// TwinCAT 3 PLC project TcoCognexVision
// Title: TcoCognexVision
// Company: Vortex.Library
// ProjectVersion: 0.6.0.913
// ProgramVersion: 3.1.4023.0
// libraries:
//   Tc2_Standard, * (Beckhoff Automation GmbH)
//   Tc2_System, * (Beckhoff Automation GmbH)
//   Tc3_Module, * (Beckhoff Automation GmbH)
//   TcoAbstractions, 0.6.0.913 (Vortex.Library)
//   TcoCore, 0.6.0.913 (Vortex.Library)
//   TcoIo, 0.6.0.913 (Vortex.Library)
//   TcoUtilities, 0.6.0.913 (Vortex.Library)
// project tree:
//   / PlcTask.TcTTO
//   POUs/TcoDataman/v_5_x_x/IO/ TcoDatamanAcquisitionControl_v_5_x_x.TcDUT, TcoDatamanAcquisitionStatus_v_5_x_x.TcDUT, TcoDatamanIO_v_5_x_x.TcDUT, TcoDatamanResultData_v_5_x_x.TcDUT, TcoDatamanResultsControl_v_5_x_x.TcDUT, TcoDatamanResultsStatus_v_5_x_x.TcDUT, TcoDatamanSoftEventControl_v_5_x_x.TcDUT, TcoDatamanUserData_v_5_x_x.TcDUT
//   POUs/TcoDataman/v_5_x_x/Structs/ eDatamanResultDataSize_v_5_x_x.TcDUT, eDatamanUserDataSize_v_5_x_x.TcDUT, TcoDatamanConfig_v_5_x_x.TcDUT, TcoDatamanResults_v_5_x_x.TcDUT, TcoDatamanSignalStates_v_5_x_x.TcDUT, TcoDatamanStatus_v_5_x_x.TcDUT, TcoDatamanUser_v_5_x_x.TcDUT
//   POUs/TcoDataman/v_5_x_x/Tasks/ TcoDatamanClearResultData_v_5_x_x.TcPOU, TcoDatamanRead_v_5_x_x.TcPOU
//   POUs/TcoDataman/v_5_x_x/ TcoDataman_v_5_x_x.TcPOU
//   POUs/TcoDesigner/Structs/ eTcoDesignerTriggerType.TcDUT, TcoDesignerConfig_v_2_x_x.TcDUT, TcoDesignerData_2_x_x.TcDUT, TcoDesignerRootContainer.TcPOU, TcoDesignerStatus_v_2_x_x.TcDUT, TcoDesignerGenericResults_v_2_x_x.TcDUT, TcoDesignerPcToPlc_v_2_x_x.TcDUT, TcoDesignerPlcToPc_v_2_x_x.TcDUT
//   POUs/TcoDesigner/Tasks/ TcoDesignerTrigger_v_2_x_x.TcPOU, TcoDesignerClearInspectionResults_v_2_x_x.TcPOU
//   POUs/TcoDesigner/ TcoDesigner_v_2_x_x.TcPOU
//   POUs/TcoInsight/v_5_x_x/IO/ TcoInsightAcquisitionControl_v_5_x_x.TcDUT, TcoInsightAcquisitionStatus_v_5_x_x.TcDUT, TcoInsightIO_v_5_x_x.TcDUT, TcoInsightResultData_v_5_x_x.TcDUT, TcoInsightInspectionControl_v_5_x_x.TcDUT, TcoInsightInspectionStatus_v_5_x_x.TcDUT, TcoInsightSoftEventControl_v_5_x_x.TcDUT, TcoInsightCommandControl_v_5_x_x.TcDUT, TcoInsightUserData_v_5_x_x.TcDUT
//   POUs/TcoInsight/v_5_x_x/Structs/ eTcoInsightResultDataSize_v_5_x_x.TcDUT, eTcoInsightUserDataSize_v_5_x_x.TcDUT, TcoInsightConfig_v_5_x_x.TcDUT, TcoInsightResults_v_5_x_x.TcDUT, TcoInsightSignalStates_v_5_x_x.TcDUT, TcoInsightStatus_v_5_x_x.TcDUT, TcoInsightUser_v_5_x_x.TcDUT
//   POUs/TcoInsight/v_5_x_x/Tasks/ TcoInsightTrigger_v_5_x_x.TcPOU, TcoInsightChangeJobByName_v_5_x_x.TcPOU, TcoInsightChangeJobByNumber_v_5_x_x.TcPOU, TcoInsightClearInspectionResults_v_5_x_x.TcPOU, TcoInsightSoftEvent_v_5_x_x.TcPOU
//   POUs/TcoInsight/v_5_x_x/ TcoInsight_v_5_x_x.TcPOU
//   POUs/ TcoVisionParams.TcGVL
// real-time tasks:
//   TASK PlcTask: cycle T#10ms, priority 20, ADS port 350
//   TASK PNIO: cycle T#8ms, priority 21, ADS port 351
// I/O:
//   DEVICE Device 1 (Profinet Controller) (disabled), AmsNetId 172.20.10.104.2.1
//     dm260 [Cognex DataMan 260 ID Reader DMR-260#-#0]
//       modules: DAP_Module, Acquisition_Control, Acquisition_Status, Results_Control, Results_Status, Soft_Event_Control, User_Data_64_bytes, Result_Data_64_bytes
//     dm8700 [Cognex DataMan 8700 ID Reader CC-B DMR-87xx-xx]
//       modules: DAP_Module, Acquisition_Control, Acquisition_Status, Results_Control, Results_Status, Soft_Event_Control, User_Data_64_bytes, Result_Data_64_bytes
// variable links:
//   TcoCognexVision/TcoCognexVision Instance <-> Device 1 (Profinet Controller)/dm260
//     PlcTask Inputs/IO.dm260.AcquisitionStatus.Acquiring <-> API/Acquisition_Status/Acquisition_Status/Inputs/Acquisition_Status_Register/Acquiring
//     PlcTask Inputs/IO.dm260.AcquisitionStatus.MissedAcquisition <-> API/Acquisition_Status/Acquisition_Status/Inputs/Acquisition_Status_Register/Missed_Acquisition
//     PlcTask Inputs/IO.dm260.AcquisitionStatus.TriggerAcknowledge <-> API/Acquisition_Status/Acquisition_Status/Inputs/Acquisition_Status_Register/Trigger_Acknowledge
//     PlcTask Inputs/IO.dm260.AcquisitionStatus.TriggerID <-> API/Acquisition_Status/Acquisition_Status/Inputs/Trigger_ID
//     PlcTask Inputs/IO.dm260.AcquisitionStatus.TriggerReady <-> API/Acquisition_Status/Acquisition_Status/Inputs/Acquisition_Status_Register/Trigger_Ready
//     PlcTask Inputs/IO.dm260.PnIoBoxDiag <-> Inputs/PnIoBoxDiag
//     PlcTask Inputs/IO.dm260.PnIoBoxState <-> Inputs/PnIoBoxState
//     PlcTask Inputs/IO.dm260.ResultData.ResultCode <-> API/Result_Data_64_bytes/Result_Data_64_bytes/Inputs/Result_Code
//     PlcTask Inputs/IO.dm260.ResultData.ResultData <-> API/Result_Data_64_bytes/Result_Data_64_bytes/Inputs/Result_Data
//     PlcTask Inputs/IO.dm260.ResultData.ResultExtended <-> API/Result_Data_64_bytes/Result_Data_64_bytes/Inputs/Result_Extended
//     PlcTask Inputs/IO.dm260.ResultData.ResultID <-> API/Result_Data_64_bytes/Result_Data_64_bytes/Inputs/Result_ID
//     PlcTask Inputs/IO.dm260.ResultData.ResultLength <-> API/Result_Data_64_bytes/Result_Data_64_bytes/Inputs/Result_Length
//     PlcTask Inputs/IO.dm260.ResultsStatus.DecodeComplete <-> API/Results_Status/Results_Status/Inputs/Results_Status_Register/Decode_Complete
//     PlcTask Inputs/IO.dm260.ResultsStatus.Decoding <-> API/Results_Status/Results_Status/Inputs/Results_Status_Register/Decoding
//     PlcTask Inputs/IO.dm260.ResultsStatus.ErrorDetected <-> API/Results_Status/Results_Status/Inputs/Results_Status_Register/Set_when_reader_fault_occurs
//     PlcTask Inputs/IO.dm260.ResultsStatus.ResultsAvailable <-> API/Results_Status/Results_Status/Inputs/Results_Status_Register/Results_Available
//     PlcTask Inputs/IO.dm260.ResultsStatus.ResultsBufferOverrun <-> API/Results_Status/Results_Status/Inputs/Results_Status_Register/Results_Buffer_Overrun
//     PlcTask Inputs/IO.dm260.SoftEventControl.ExecuteDMCCAcknowledge <-> API/Soft_Event_Control/Soft_Event_Control/Inputs/Soft_Event_Acknowledge_Register/Execute_DMCC_Acknowledge
//     PlcTask Inputs/IO.dm260.SoftEventControl.SetMatchStringAcknowledge <-> API/Soft_Event_Control/Soft_Event_Control/Inputs/Soft_Event_Acknowledge_Register/Set_Match_String_Acknowledge
//     PlcTask Inputs/IO.dm260.SoftEventControl.TrainBrightnessAcknowledge <-> API/Soft_Event_Control/Soft_Event_Control/Inputs/Soft_Event_Acknowledge_Register/Train_Brightness_Acknowledge
//     PlcTask Inputs/IO.dm260.SoftEventControl.TrainCodeAcknowledge <-> API/Soft_Event_Control/Soft_Event_Control/Inputs/Soft_Event_Acknowledge_Register/Train_Code_Acknowledge
//     PlcTask Inputs/IO.dm260.SoftEventControl.TrainFocusAcknowledge <-> API/Soft_Event_Control/Soft_Event_Control/Inputs/Soft_Event_Acknowledge_Register/Train_Focus_Acknowledge
//     PlcTask Inputs/IO.dm260.SoftEventControl.TrainMatchStringAcknowledge <-> API/Soft_Event_Control/Soft_Event_Control/Inputs/Soft_Event_Acknowledge_Register/Train_Match_String_Acknowledge
//     PlcTask Inputs/IO.dm260.SoftEventControl.UntrainAcknowledge <-> API/Soft_Event_Control/Soft_Event_Control/Inputs/Soft_Event_Acknowledge_Register/Untrain_Acknowledge
//     PlcTask Outputs/IO.dm260.AcquisitionControl.Trigger <-> API/Acquisition_Control/Acquisition_Control/Outputs/Acquisition_Control_Register/Trigger
//     PlcTask Outputs/IO.dm260.AcquisitionControl.TriggerEnable <-> API/Acquisition_Control/Acquisition_Control/Outputs/Acquisition_Control_Register/Trigger_Enable
//     PlcTask Outputs/IO.dm260.PnIoBoxCtrl <-> Outputs/PnIoBoxCtrl
//     PlcTask Outputs/IO.dm260.ResultsControl.EnableResultBuffering <-> API/Results_Control/Results_Control/Outputs/Results_Control_Register/Enable_Result_Buffering
//     PlcTask Outputs/IO.dm260.ResultsControl.ResultsAcknowledge <-> API/Results_Control/Results_Control/Outputs/Results_Control_Register/Results_Acknowledge
//     PlcTask Outputs/IO.dm260.SoftEventControl.ExecuteDMCC <-> API/Soft_Event_Control/Soft_Event_Control/Outputs/Soft_Event_Control_Register/Execute_DMCC
//     PlcTask Outputs/IO.dm260.SoftEventControl.SetMatchString <-> API/Soft_Event_Control/Soft_Event_Control/Outputs/Soft_Event_Control_Register/Set_Match_String
//     PlcTask Outputs/IO.dm260.SoftEventControl.TrainBrightness <-> API/Soft_Event_Control/Soft_Event_Control/Outputs/Soft_Event_Control_Register/Train_Brightness
//     PlcTask Outputs/IO.dm260.SoftEventControl.TrainCode <-> API/Soft_Event_Control/Soft_Event_Control/Outputs/Soft_Event_Control_Register/Train_Code
//     PlcTask Outputs/IO.dm260.SoftEventControl.TrainFocus <-> API/Soft_Event_Control/Soft_Event_Control/Outputs/Soft_Event_Control_Register/Train_Focus
//     PlcTask Outputs/IO.dm260.SoftEventControl.TrainMatchString <-> API/Soft_Event_Control/Soft_Event_Control/Outputs/Soft_Event_Control_Register/Train_Match_String
//     PlcTask Outputs/IO.dm260.SoftEventControl.Untrain <-> API/Soft_Event_Control/Soft_Event_Control/Outputs/Soft_Event_Control_Register/Untrain
//     PlcTask Outputs/IO.dm260.UserData.UserData <-> API/User_Data_64_bytes/User_Data_64_bytes/Outputs/User_Data
//     PlcTask Outputs/IO.dm260.UserData.UserDataLength <-> API/User_Data_64_bytes/User_Data_64_bytes/Outputs/User_Data_Length
//     PlcTask Outputs/IO.dm260.UserData.UserDataOption <-> API/User_Data_64_bytes/User_Data_64_bytes/Outputs/User_Data_Option
//   TcoCognexVision/TcoCognexVision Instance <-> Device 1 (Profinet Controller)/dm8700
//     PlcTask Inputs/IO.dm8700.AcquisitionStatus.Acquiring <-> API/Acquisition_Status/Acquisition_Status/Inputs/Acquisition_Status_Register/Acquiring
//     PlcTask Inputs/IO.dm8700.AcquisitionStatus.MissedAcquisition <-> API/Acquisition_Status/Acquisition_Status/Inputs/Acquisition_Status_Register/Missed_Acquisition
//     PlcTask Inputs/IO.dm8700.AcquisitionStatus.TriggerAcknowledge <-> API/Acquisition_Status/Acquisition_Status/Inputs/Acquisition_Status_Register/Trigger_Acknowledge
//     PlcTask Inputs/IO.dm8700.AcquisitionStatus.TriggerID <-> API/Acquisition_Status/Acquisition_Status/Inputs/Trigger_ID
//     PlcTask Inputs/IO.dm8700.AcquisitionStatus.TriggerReady <-> API/Acquisition_Status/Acquisition_Status/Inputs/Acquisition_Status_Register/Trigger_Ready
//     PlcTask Inputs/IO.dm8700.PnIoBoxDiag <-> Inputs/PnIoBoxDiag
//     PlcTask Inputs/IO.dm8700.PnIoBoxState <-> Inputs/PnIoBoxState
//     PlcTask Inputs/IO.dm8700.ResultData.ResultCode <-> API/Result_Data_64_bytes/Result_Data_64_bytes/Inputs/Result_Code
//     PlcTask Inputs/IO.dm8700.ResultData.ResultData <-> API/Result_Data_64_bytes/Result_Data_64_bytes/Inputs/Result_Data
//     PlcTask Inputs/IO.dm8700.ResultData.ResultExtended <-> API/Result_Data_64_bytes/Result_Data_64_bytes/Inputs/Result_Extended
//     PlcTask Inputs/IO.dm8700.ResultData.ResultID <-> API/Result_Data_64_bytes/Result_Data_64_bytes/Inputs/Result_ID
//     PlcTask Inputs/IO.dm8700.ResultData.ResultLength <-> API/Result_Data_64_bytes/Result_Data_64_bytes/Inputs/Result_Length
//     PlcTask Inputs/IO.dm8700.ResultsStatus.DecodeComplete <-> API/Results_Status/Results_Status/Inputs/Results_Status_Register/Decode_Complete
//     PlcTask Inputs/IO.dm8700.ResultsStatus.Decoding <-> API/Results_Status/Results_Status/Inputs/Results_Status_Register/Decoding
//     PlcTask Inputs/IO.dm8700.ResultsStatus.ErrorDetected <-> API/Results_Status/Results_Status/Inputs/Results_Status_Register/Set_when_reader_fault_occurs
//     PlcTask Inputs/IO.dm8700.ResultsStatus.ResultsAvailable <-> API/Results_Status/Results_Status/Inputs/Results_Status_Register/Results_Available
//     PlcTask Inputs/IO.dm8700.ResultsStatus.ResultsBufferOverrun <-> API/Results_Status/Results_Status/Inputs/Results_Status_Register/Results_Buffer_Overrun
//     PlcTask Inputs/IO.dm8700.SoftEventControl.ExecuteDMCCAcknowledge <-> API/Soft_Event_Control/Soft_Event_Control/Inputs/Soft_Event_Acknowledge_Register/Execute_DMCC_Acknowledge
//     PlcTask Inputs/IO.dm8700.SoftEventControl.SetMatchStringAcknowledge <-> API/Soft_Event_Control/Soft_Event_Control/Inputs/Soft_Event_Acknowledge_Register/Set_Match_String_Acknowledge
//     PlcTask Inputs/IO.dm8700.SoftEventControl.TrainBrightnessAcknowledge <-> API/Soft_Event_Control/Soft_Event_Control/Inputs/Soft_Event_Acknowledge_Register/Train_Brightness_Acknowledge
//     PlcTask Inputs/IO.dm8700.SoftEventControl.TrainCodeAcknowledge <-> API/Soft_Event_Control/Soft_Event_Control/Inputs/Soft_Event_Acknowledge_Register/Train_Code_Acknowledge
//     PlcTask Inputs/IO.dm8700.SoftEventControl.TrainFocusAcknowledge <-> API/Soft_Event_Control/Soft_Event_Control/Inputs/Soft_Event_Acknowledge_Register/Train_Focus_Acknowledge
//     PlcTask Inputs/IO.dm8700.SoftEventControl.TrainMatchStringAcknowledge <-> API/Soft_Event_Control/Soft_Event_Control/Inputs/Soft_Event_Acknowledge_Register/Train_Match_String_Acknowledge
//     PlcTask Inputs/IO.dm8700.SoftEventControl.UntrainAcknowledge <-> API/Soft_Event_Control/Soft_Event_Control/Inputs/Soft_Event_Acknowledge_Register/Untrain_Acknowledge
//     PlcTask Outputs/IO.dm8700.AcquisitionControl.Trigger <-> API/Acquisition_Control/Acquisition_Control/Outputs/Acquisition_Control_Register/Trigger
//     PlcTask Outputs/IO.dm8700.AcquisitionControl.TriggerEnable <-> API/Acquisition_Control/Acquisition_Control/Outputs/Acquisition_Control_Register/Trigger_Enable
//     PlcTask Outputs/IO.dm8700.PnIoBoxCtrl <-> Outputs/PnIoBoxCtrl
//     PlcTask Outputs/IO.dm8700.ResultsControl.EnableResultBuffering <-> API/Results_Control/Results_Control/Outputs/Results_Control_Register/Enable_Result_Buffering
//     PlcTask Outputs/IO.dm8700.ResultsControl.ResultsAcknowledge <-> API/Results_Control/Results_Control/Outputs/Results_Control_Register/Results_Acknowledge
//     PlcTask Outputs/IO.dm8700.SoftEventControl.ExecuteDMCC <-> API/Soft_Event_Control/Soft_Event_Control/Outputs/Soft_Event_Control_Register/Execute_DMCC
//     PlcTask Outputs/IO.dm8700.SoftEventControl.SetMatchString <-> API/Soft_Event_Control/Soft_Event_Control/Outputs/Soft_Event_Control_Register/Set_Match_String
//     PlcTask Outputs/IO.dm8700.SoftEventControl.TrainBrightness <-> API/Soft_Event_Control/Soft_Event_Control/Outputs/Soft_Event_Control_Register/Train_Brightness
//     PlcTask Outputs/IO.dm8700.SoftEventControl.TrainCode <-> API/Soft_Event_Control/Soft_Event_Control/Outputs/Soft_Event_Control_Register/Train_Code
//     PlcTask Outputs/IO.dm8700.SoftEventControl.TrainFocus <-> API/Soft_Event_Control/Soft_Event_Control/Outputs/Soft_Event_Control_Register/Train_Focus
//     PlcTask Outputs/IO.dm8700.SoftEventControl.TrainMatchString <-> API/Soft_Event_Control/Soft_Event_Control/Outputs/Soft_Event_Control_Register/Train_Match_String
//     PlcTask Outputs/IO.dm8700.SoftEventControl.Untrain <-> API/Soft_Event_Control/Soft_Event_Control/Outputs/Soft_Event_Control_Register/Untrain
//     PlcTask Outputs/IO.dm8700.UserData.UserData <-> API/User_Data_64_bytes/User_Data_64_bytes/Outputs/User_Data
//     PlcTask Outputs/IO.dm8700.UserData.UserDataLength <-> API/User_Data_64_bytes/User_Data_64_bytes/Outputs/User_Data_Length
//     PlcTask Outputs/IO.dm8700.UserData.UserDataOption <-> API/User_Data_64_bytes/User_Data_64_bytes/Outputs/User_Data_Option

CONFIGURATION TcoCognexVision
    RESOURCE PLC ON TwinCAT3
        TASK PlcTask(INTERVAL := T#10ms, PRIORITY := 20);
        PROGRAM MAIN WITH PlcTask : MAIN;
    END_RESOURCE
END_CONFIGURATION

// ---- POUs/TcoDataman/v_5_x_x/IO/TcoDatamanAcquisitionControl_v_5_x_x.TcDUT
TYPE TcoDatamanAcquisitionControl_v_5_x_x :
STRUCT
    TriggerEnable AT %Q* : BOOL;
    Trigger AT %Q* : BOOL;
END_STRUCT
END_TYPE

// ---- POUs/TcoDataman/v_5_x_x/IO/TcoDatamanAcquisitionStatus_v_5_x_x.TcDUT
TYPE TcoDatamanAcquisitionStatus_v_5_x_x :
STRUCT
    TriggerReady AT %I* : BOOL;
    TriggerAcknowledge AT %I* : BOOL;
    Acquiring AT %I* : BOOL;
    MissedAcquisition AT %I* : BOOL;
    TriggerID AT %I* : UINT;
END_STRUCT
END_TYPE

// ---- POUs/TcoDataman/v_5_x_x/IO/TcoDatamanIO_v_5_x_x.TcDUT
TYPE TcoDatamanIO_v_5_x_x :
STRUCT
    PnIoBoxState AT %I* : UINT;
    PnIoBoxDiag AT %I* : UINT;
    PnIoBoxCtrl AT %Q* : UINT;
    AcquisitionControl : TcoDatamanAcquisitionControl_v_5_x_x;
    AcquisitionStatus : TcoDatamanAcquisitionStatus_v_5_x_x;
    ResultsControl : TcoDatamanResultsControl_v_5_x_x;
    ResultsStatus : TcoDatamanResultsStatus_v_5_x_x;
    SoftEventControl : TcoDatamanSoftEventControl_v_5_x_x;
    UserData : TcoDatamanUserData_v_5_x_x;
    ResultData : TcoDatamanResultData_v_5_x_x;
END_STRUCT
END_TYPE

// ---- POUs/TcoDataman/v_5_x_x/IO/TcoDatamanResultData_v_5_x_x.TcDUT
TYPE TcoDatamanResultData_v_5_x_x :
STRUCT
    ResultID AT %I* : UINT;
    ResultCode AT %I* : UINT;
    ResultExtended AT %I* : UINT;
    ResultLength AT %I* : UINT;
    ResultData AT %I* : ARRAY[0..245] OF BYTE;
END_STRUCT
END_TYPE

// ---- POUs/TcoDataman/v_5_x_x/IO/TcoDatamanResultsControl_v_5_x_x.TcDUT
TYPE TcoDatamanResultsControl_v_5_x_x :
STRUCT
    EnableResultBuffering AT %Q* : BOOL;
    ResultsAcknowledge AT %Q* : BOOL;
END_STRUCT
END_TYPE

// ---- POUs/TcoDataman/v_5_x_x/IO/TcoDatamanResultsStatus_v_5_x_x.TcDUT
TYPE TcoDatamanResultsStatus_v_5_x_x :
STRUCT
    Decoding AT %I* : BOOL;
    DecodeComplete AT %I* : BOOL;
    ResultsBufferOverrun AT %I* : BOOL;
    ResultsAvailable AT %I* : BOOL;
    ErrorDetected AT %I* : BOOL;
END_STRUCT
END_TYPE

// ---- POUs/TcoDataman/v_5_x_x/IO/TcoDatamanSoftEventControl_v_5_x_x.TcDUT
TYPE TcoDatamanSoftEventControl_v_5_x_x :
STRUCT
    TrainCodeAcknowledge AT %I* : BOOL;
    TrainMatchStringAcknowledge AT %I* : BOOL;
    TrainFocusAcknowledge AT %I* : BOOL;
    TrainBrightnessAcknowledge AT %I* : BOOL;
    UntrainAcknowledge AT %I* : BOOL;
    Reserved05 AT %I* : BOOL;
    ExecuteDMCCAcknowledge AT %I* : BOOL;
    SetMatchStringAcknowledge AT %I* : BOOL;
    TrainCode AT %Q* : BOOL;
    TrainMatchString AT %Q* : BOOL;
    TrainFocus AT %Q* : BOOL;
    TrainBrightness AT %Q* : BOOL;
    Untrain AT %Q* : BOOL;
    Reserved15 AT %Q* : BOOL;
    ExecuteDMCC AT %Q* : BOOL;
    SetMatchString AT %Q* : BOOL;
END_STRUCT
END_TYPE

// ---- POUs/TcoDataman/v_5_x_x/IO/TcoDatamanUserData_v_5_x_x.TcDUT
TYPE TcoDatamanUserData_v_5_x_x :
STRUCT
    UserDataOption AT %Q* : UINT;
    UserDataLength AT %Q* : UINT;
    UserData AT %Q* : ARRAY[0..249] OF BYTE;
END_STRUCT
END_TYPE

// ---- POUs/TcoDataman/v_5_x_x/Structs/eDatamanResultDataSize_v_5_x_x.TcDUT
{attribute 'qualified_only'}
{attribute 'strict'}
TYPE eDatamanResultDataSize_v_5_x_x :
(
    RESULT_DATA_16B := 16,
    RESULT_DATA_32B := 32,
    RESULT_DATA_64B := 64,
    RESULT_DATA_128B := 128,
    RESULT_DATA_246B := 246
);
END_TYPE

// ---- POUs/TcoDataman/v_5_x_x/Structs/eDatamanUserDataSize_v_5_x_x.TcDUT
{attribute 'qualified_only'}
{attribute 'strict'}
TYPE eDatamanUserDataSize_v_5_x_x :
(
    USER_DATA_16B := 16,
    USER_DATA_32B := 32,
    USER_DATA_64B := 64,
    USER_DATA_128B := 128,
    USER_DATA_250B := 250
);
END_TYPE

// ---- POUs/TcoDataman/v_5_x_x/Structs/TcoDatamanConfig_v_5_x_x.TcDUT
TYPE TcoDatamanConfig_v_5_x_x :
STRUCT
    ResultDataSize : eDatamanResultDataSize_v_5_x_x := eDatamanResultDataSize_v_5_x_x.RESULT_DATA_64B;
    UserDataSize : eDatamanUserDataSize_v_5_x_x := eDatamanUserDataSize_v_5_x_x.USER_DATA_64B;
    DataFormat : eTcoDataFormat := TcoUtilities.eTcoDataFormat.BigEndian;
    ContinuousReading : BOOL := FALSE;
    UpdateStatesPermanently : BOOL := FALSE;
    InfoTime : TIME := T#2S;
    ErrorTime : TIME := T#5S;
    ShowUserData : BOOL := FALSE;
    ShowResultsData : BOOL := FALSE;
END_STRUCT
END_TYPE

// ---- POUs/TcoDataman/v_5_x_x/Structs/TcoDatamanResults_v_5_x_x.TcDUT
TYPE TcoDatamanResults_v_5_x_x :
STRUCT
    Id : UINT;
    Code : UINT;
    Extended : UINT;
    Length : UINT;
    Data : ARRAY[0..TcoVisionParams.MAX_BYTE_ARRAY] OF BYTE;
END_STRUCT
END_TYPE

// ---- POUs/TcoDataman/v_5_x_x/Structs/TcoDatamanSignalStates_v_5_x_x.TcDUT
{attribute addProperty Name "Signal states"}
{attribute wpf [Container(Layout.Stack)]}
TYPE TcoDatamanSignalStates_v_5_x_x :
STRUCT
    {attribute wpf [Container(Layout.Stack,"Acquisition control")]}
    {attribute wpf [Group(Layout.GroupBox)]}
    {attribute addProperty Name "<#Trigger enable#>"}
    TriggerEnable : BOOL;
    {attribute addProperty Name "<#Trigger#>"}
    Trigger : BOOL;
    {attribute wpf [Container(Layout.Stack,"Result control")]}
    {attribute wpf [Group(Layout.GroupBox)]}
    {attribute addProperty Name "<#Enable result buffering#>"}
    EnableResultBuffering : BOOL;
    {attribute addProperty Name "<#Result acknowledge#>"}
    ResultsAcknowledge : BOOL;
    {attribute wpf [Container(Layout.Stack,"Acquisition status")]}
    {attribute wpf [Group(Layout.GroupBox)]}
    {attribute addProperty Name "<#Trigger ready#>"}
    TriggerReady : BOOL;
    {attribute addProperty Name "<#Trigger acknowledge#>"}
    TriggerAcknowledge : BOOL;
    {attribute addProperty Name "<#Acquiring#>"}
    Acquiring : BOOL;
    {attribute addProperty Name "<#Missed acquisition#>"}
    MissedAcquisition : BOOL;
    {attribute addProperty Name "<#Trigger ID#>"}
    TriggerID : UINT;
    {attribute wpf [Container(Layout.Stack,"Result status")]}
    {attribute wpf [Group(Layout.GroupBox)]}
    {attribute addProperty Name "<#Decoding#>"}
    Decoding : BOOL;
    {attribute addProperty Name "<#Decode complete#>"}
    DecodeComplete : BOOL;
    {attribute addProperty Name "<#Result buffer overrun#>"}
    ResultsBufferOverrun : BOOL;
    {attribute addProperty Name "<#Results available#>"}
    ResultsAvailable : BOOL;
    {attribute addProperty Name "<#Error detected#>"}
    ErrorDetected : BOOL;
    {attribute wpf [Container(Layout.Stack,"Result data")]}
    {attribute wpf [Group(Layout.GroupBox)]}
    {attribute addProperty Name "<#Result ID#>"}
    ResultID : UINT;
    {attribute addProperty Name "<#Result code#>"}
    ResultCode : UINT;
    {attribute addProperty Name "<#Result extended#>"}
    ResultExtended : UINT;
    {attribute addProperty Name "<#Result length#>"}
    ResultLength : UINT;
END_STRUCT
END_TYPE

// ---- POUs/TcoDataman/v_5_x_x/Structs/TcoDatamanStatus_v_5_x_x.TcDUT
TYPE TcoDatamanStatus_v_5_x_x :
STRUCT
    ActionDescription : STRING(100);
    ResultString : STRING;
    SignalStatus : TcoDatamanSignalStates_v_5_x_x;
END_STRUCT
END_TYPE

// ---- POUs/TcoDataman/v_5_x_x/Structs/TcoDatamanUser_v_5_x_x.TcDUT
TYPE TcoDatamanUser_v_5_x_x :
STRUCT
    Option : UINT;
    Length : UINT;
    Data : ARRAY[0..TcoVisionParams.MAX_BYTE_ARRAY] OF BYTE;
END_STRUCT
END_TYPE

// ---- POUs/TcoDesigner/Structs/eTcoDesignerTriggerType.TcDUT
{attribute 'qualified_only'}
{attribute 'strict'}
TYPE eTcoDesignerTriggerType :
(
    Trigger := 0,
    TriggerFast := 1,
    TriggerWithTimeout := 2
);
END_TYPE

// ---- POUs/TcoDesigner/Structs/TcoDesignerConfig_v_2_x_x.TcDUT
TYPE TcoDesignerConfig_v_2_x_x :
STRUCT
    TriggerTimemout : TIME := T#15S;
    ConnectionTimemout : TIME := T#10S;
    InfoTime : TIME := T#2S;
    ErrorTime : TIME := T#5S;
END_STRUCT
END_TYPE

// ---- POUs/TcoDesigner/Structs/TcoDesignerData_2_x_x.TcDUT
{attribute wpf [Container(Layout.Stack)]}
TYPE TcoDesignerData_2_x_x :
STRUCT
    {attribute wpf [Container(Layout.Stack,"PcToPlc")]}
    {attribute addProperty Name "<#PCtoPLC#>"}
    PcToPlc : TcoDesignerPcToPlc_v_2_x_x;
    {attribute wpf [Container(Layout.Stack,"PlcToPc")]}
    {attribute addProperty Name "<#PLCtoPC#>"}
    PlcToPc : TcoDesignerPlcToPc_v_2_x_x;
END_STRUCT
END_TYPE

// ---- POUs/TcoDesigner/Structs/TcoDesignerStatus_v_2_x_x.TcDUT
TYPE TcoDesignerStatus_v_2_x_x :
STRUCT
    ActionDescription : STRING(100);
    ClientConnected : BOOL;
    {attribute wpf [Container(Layout.Stack,"PcToPlc")]}
    {attribute wpf [Group(Layout.GroupBox)]}
    SignalStatus : TcoDesignerPcToPlc_v_2_x_x;
END_STRUCT
END_TYPE

// ---- POUs/TcoDesigner/Structs/TcoDesignerGenericResults_v_2_x_x.TcDUT
TYPE TcoDesignerGenericResults_v_2_x_x :
STRUCT
    {attribute addProperty Name "<#GeneralResult Pass#>"}
    ResultPass : BOOL;
    {attribute addProperty Name "<#GeneralResult FAIL#>"}
    ResultFail : BOOL;
END_STRUCT
END_TYPE

// ---- POUs/TcoDesigner/Structs/TcoDesignerPcToPlc_v_2_x_x.TcDUT
{attribute wpf [Container(Layout.Stack)]}
TYPE TcoDesignerPcToPlc_v_2_x_x :
STRUCT
    {attribute wpf [Container(Layout.Stack,"State")]}
    {attribute addProperty Name "<#SystemOnline#>"}
    SystemOnline : BOOL; //indication that designer PC app and inspection are running
    {attribute addProperty Name "<#InspectionReady#>"}
    InspectionReady : BOOL; // inspection is ready
    {attribute addProperty Name "<#ResultsAvailable#>"}
    ResultsAvailable : BOOL; //results are available and valid
    {attribute addProperty Name "<#JobId#>"}
    JobId : UINT; // actual job id
    {attribute addProperty Name "<#JobName#>"}
    JobName : STRING; //aktual job name
    {attribute addProperty Name "<#JobLoadDone#>"}
    JobLoadDone : BOOL;
    {attribute addProperty Name "<#ClearResultsAck#>"}
    ClearResultsAck : BOOL;
    {attribute addProperty Name "<#Trigger Counter#>"}
    TriggerCounter : UDINT;
    {attribute addProperty Name "<#Error#>"}
    Error : BOOL;
    {attribute addProperty Name "<#LiveBit#>"}
    LiveBit : BOOL;
    {attribute addProperty Name "<#ErrorMsg#>"}
    ErrorMsg : STRING;
    {attribute addProperty Name "<#TriggerTimeout#>"}
    TriggerTimeout : BOOL;
    {attribute wpf [Container(Layout.Stack,"Results")]}
    {attribute addProperty Name "<#Results#>"}
    InspectionResults : TcoDesignerGenericResults_v_2_x_x;
END_STRUCT
END_TYPE

// ---- POUs/TcoDesigner/Structs/TcoDesignerPlcToPc_v_2_x_x.TcDUT
{attribute wpf [Container(Layout.Stack)]}
TYPE TcoDesignerPlcToPc_v_2_x_x :
STRUCT
    {attribute wpf [Container(Layout.Stack,"Control")]}
    {attribute addProperty Name "<#Trigger#>"}
    Trigger : BOOL;
    {attribute addProperty Name "<#ResultsAck#>"}
    ResultsAck : BOOL;
    {attribute addProperty Name "<#Reset#>"}
    Reset : BOOL;
    {attribute addProperty Name "<#JobLoadId#>"}
    JobLoadId : UINT;
    {attribute addProperty Name "<#LoadJob#>"}
    LoadJob : BOOL;
    {attribute addProperty Name "<#ClearResults#>"}
    ClearResults : BOOL;
    {attribute addProperty Name "<#Timeout[ms]#>"}
    Timeout : UINT;
    {attribute addProperty Name "<# PartId #>"}
    PartId : STRING; //napr. DMC Code
END_STRUCT
END_TYPE

// ---- POUs/TcoInsight/v_5_x_x/IO/TcoInsightAcquisitionControl_v_5_x_x.TcDUT
TYPE TcoInsightAcquisitionControl_v_5_x_x :
STRUCT
    AcquisitionTriggerEnable AT %Q* : BOOL;
    AcquisitionTrigger AT %Q* : BOOL;
    ClearExposureComplete AT %Q* : BOOL;
    SetOffline AT %Q* : BOOL;
END_STRUCT
END_TYPE

// ---- POUs/TcoInsight/v_5_x_x/IO/TcoInsightAcquisitionStatus_v_5_x_x.TcDUT
TYPE TcoInsightAcquisitionStatus_v_5_x_x :
STRUCT
    AcquisitionTriggerReady AT %I* : BOOL;
    AcquisitionTriggerAcknowledge AT %I* : BOOL;
    ExposureComplete AT %I* : BOOL;
    MissedAcquisition AT %I* : BOOL;
    OfflineReason0 AT %I* : BOOL;
    OfflineReason1 AT %I* : BOOL;
    OfflineReason2 AT %I* : BOOL;
    Online AT %I* : BOOL;
    AcquisitionID AT %I* : UINT;
END_STRUCT
END_TYPE

// ---- POUs/TcoInsight/v_5_x_x/IO/TcoInsightIO_v_5_x_x.TcDUT
TYPE TcoInsightIO_v_5_x_x :
STRUCT
    PnIoBoxState AT %I* : UINT;
    PnIoBoxDiag AT %I* : UINT;
    PnIoBoxCtrl AT %Q* : UINT;
    AcquisitionControl : TcoInsightAcquisitionControl_v_5_x_x;
    AcquisitionStatus : TcoInsightAcquisitionStatus_v_5_x_x;
    InspectionControl : TcoInsightInspectionControl_v_5_x_x;
    InspectionStatus : TcoInsightInspectionStatus_v_5_x_x;
    CommandControl : TcoInsightCommandControl_v_5_x_x;
    SoftEventControl : TcoInsightSoftEventControl_v_5_x_x;
    UserData : TcoInsightUserData_v_5_x_x;
    ResultsData : TcoInsightResultData_v_5_x_x;
END_STRUCT
END_TYPE

// ---- POUs/TcoInsight/v_5_x_x/IO/TcoInsightResultData_v_5_x_x.TcDUT
TYPE TcoInsightResultData_v_5_x_x :
STRUCT
    InspectionID AT %I* : UINT;
    ResultCode AT %I* : UINT;
    InspectionResults AT %I* : ARRAY[0..245] OF BYTE;
END_STRUCT
END_TYPE

// ---- POUs/TcoInsight/v_5_x_x/IO/TcoInsightInspectionControl_v_5_x_x.TcDUT
TYPE TcoInsightInspectionControl_v_5_x_x :
STRUCT
    EnableResultsBuffering AT %Q* : BOOL;
    AcknowledgeInspectionResults AT %Q* : BOOL;
    ExtendedUserDataSet AT %Q* : BOOL;
    ExecuteCommand AT %Q* : BOOL;
    ClearError AT %Q* : BOOL;
END_STRUCT
END_TYPE

// ---- POUs/TcoInsight/v_5_x_x/IO/TcoInsightInspectionStatus_v_5_x_x.TcDUT
TYPE TcoInsightInspectionStatus_v_5_x_x :
STRUCT
    SystemBusy AT %I* : BOOL;
    InspectionCompleted AT %I* : BOOL;
    ResultsBufferOverrun AT %I* : BOOL;
    ResultsValid AT %I* : BOOL;
    CommandExecuting AT %I* : BOOL;
    CommandComplete AT %I* : BOOL;
    CommandFailed AT %I* : BOOL;
    ExtendedUserDataSetAcknowledge AT %I* : BOOL;
    OverallJobPassFail AT %I* : BOOL;
    TestRunReady AT %I* : BOOL;
    Error AT %I* : BOOL;
    ErrorCode AT %I* : UINT;
END_STRUCT
END_TYPE

// ---- POUs/TcoInsight/v_5_x_x/IO/TcoInsightSoftEventControl_v_5_x_x.TcDUT
TYPE TcoInsightSoftEventControl_v_5_x_x :
STRUCT
    TriggerSoftEventAcknowledge AT %I* : ARRAY[0..7] OF BOOL;
    TriggerSoftEvent AT %Q* : ARRAY[0..7] OF BOOL;
END_STRUCT
END_TYPE

// ---- POUs/TcoInsight/v_5_x_x/IO/TcoInsightCommandControl_v_5_x_x.TcDUT
TYPE TcoInsightCommandControl_v_5_x_x :
STRUCT
    CurrentJobID AT %I* : UINT;
    Command AT %Q* : UINT;
END_STRUCT
END_TYPE

// ---- POUs/TcoInsight/v_5_x_x/IO/TcoInsightUserData_v_5_x_x.TcDUT
TYPE TcoInsightUserData_v_5_x_x :
STRUCT
    UserData AT %Q* : ARRAY[0..253] OF BYTE;
END_STRUCT
END_TYPE

// ---- POUs/TcoInsight/v_5_x_x/Structs/eTcoInsightResultDataSize_v_5_x_x.TcDUT
{attribute 'qualified_only'}
{attribute 'strict'}
TYPE eTcoInsightResultDataSize_v_5_x_x :
(
    RESULT_DATA_16B := 16,
    RESULT_DATA_32B := 32,
    RESULT_DATA_64B := 64,
    RESULT_DATA_128B := 128,
    RESULT_DATA_246B := 250
);
END_TYPE

// ---- POUs/TcoInsight/v_5_x_x/Structs/eTcoInsightUserDataSize_v_5_x_x.TcDUT
{attribute 'qualified_only'}
{attribute 'strict'}
TYPE eTcoInsightUserDataSize_v_5_x_x :
(
    USER_DATA_16B := 16,
    USER_DATA_32B := 32,
    USER_DATA_64B := 64,
    USER_DATA_128B := 128,
    USER_DATA_250B := 254
);
END_TYPE

// ---- POUs/TcoInsight/v_5_x_x/Structs/TcoInsightConfig_v_5_x_x.TcDUT
TYPE TcoInsightConfig_v_5_x_x :
STRUCT
    ResultDataSize : eTcoInsightResultDataSize_v_5_x_x := eTcoInsightResultDataSize_v_5_x_x.RESULT_DATA_64B;
    UserDataSize : eTcoInsightUserDataSize_v_5_x_x := eTcoInsightUserDataSize_v_5_x_x.USER_DATA_64B;
    DataFormat : eTcoDataFormat := TcoUtilities.eTcoDataFormat.BigEndian;
    UpdateStatesPermanently : BOOL := FALSE;
    MaxJobNumber : UINT := 999;
    InfoTime : TIME := T#2S;
    ErrorTime : TIME := T#5S;
    ShowUserData : BOOL := FALSE;
    ShowResultsData : BOOL := FALSE;
//	ServiceJobNumber		:	UINT;
//	ServiceJobName			:	STRING;
//	ServiceSoftEventNumber	:	UINT;
END_STRUCT
END_TYPE

// ---- POUs/TcoInsight/v_5_x_x/Structs/TcoInsightResults_v_5_x_x.TcDUT
TYPE TcoInsightResults_v_5_x_x :
STRUCT
    InspectionId : UINT;
    ResultCode : UINT;
    InspectionResults : ARRAY[0..TcoVisionParams.MAX_BYTE_ARRAY] OF BYTE;
END_STRUCT
END_TYPE

// ---- POUs/TcoInsight/v_5_x_x/Structs/TcoInsightSignalStates_v_5_x_x.TcDUT
{attribute addProperty Name "Signal states"}
TYPE TcoInsightSignalStates_v_5_x_x :
STRUCT
    {attribute wpf [Container(Layout.Stack,"Acquisition control")]}
    {attribute wpf [Group(Layout.GroupBox)]}
    {attribute addProperty Name "<#Acquisition trigger enable#>"}
    AcquisitionTriggerEnable : BOOL;
    {attribute addProperty Name "<#Acquisition trigger#>"}
    AcquisitionTrigger : BOOL;
    {attribute addProperty Name "<#Clear exposure complete#>"}
    ClearExposureComplete : BOOL;
    {attribute addProperty Name "<#Set offline#>"}
    SetOffline : BOOL;
    {attribute wpf [Container(Layout.Stack,"Inspection control")]}
    {attribute wpf [Group(Layout.GroupBox)]}
    {attribute addProperty Name "<#Enable results buffering#>"}
    EnableResultsBuffering AT %Q* : BOOL;
    {attribute addProperty Name "<#Acknowledge inspection results#>"}
    AcknowledgeInspectionResults AT %Q* : BOOL;
    {attribute addProperty Name "<#Extended user data set#>"}
    ExtendedUserDataSet AT %Q* : BOOL;
    {attribute addProperty Name "<#Execute command#>"}
    ExecuteCommand AT %Q* : BOOL;
    {attribute addProperty Name "<#Clear error#>"}
    ClearError AT %Q* : BOOL;
    {attribute wpf [Container(Layout.Stack,"Acquisition status")]}
    {attribute wpf [Group(Layout.GroupBox)]}
    {attribute addProperty Name "<#Acquisition trigger ready#>"}
    AcquisitionTriggerReady : BOOL;
    {attribute addProperty Name "<#Acquisition trigger acknowledge#>"}
    AcquisitionTriggerAcknowledge : BOOL;
    {attribute addProperty Name "<#Exposure complete#>"}
    ExposureComplete : BOOL;
    {attribute addProperty Name "<#Missed acquisition#>"}
    MissedAcquisition : BOOL;
    {attribute addProperty Name "<#Offline reason 0#>"}
    OfflineReason0 : BOOL;
    {attribute addProperty Name "<#Offline reason 1#>"}
    OfflineReason1 : BOOL;
    {attribute addProperty Name "<#Offline reason 2#>"}
    OfflineReason2 : BOOL;
    {attribute addProperty Name "<#Online#>"}
    Online : BOOL;
    {attribute addProperty Name "<#Acquisition ID#>"}
    AcquisitionID : UINT;
    {attribute wpf [Container(Layout.Stack,"Inspection status")]}
    {attribute wpf [Group(Layout.GroupBox)]}
    {attribute addProperty Name "<#System busy#>"}
    SystemBusy : BOOL;
    {attribute addProperty Name "<#Inspection completed#>"}
    InspectionCompleted : BOOL;
    {attribute addProperty Name "<#Results buffer overrun#>"}
    ResultsBufferOverrun : BOOL;
    {attribute addProperty Name "<#Results valid#>"}
    ResultsValid : BOOL;
    {attribute addProperty Name "<#Command executing#>"}
    CommandExecuting : BOOL;
    {attribute addProperty Name "<#Command complete#>"}
    CommandComplete : BOOL;
    {attribute addProperty Name "<#Command failed#>"}
    CommandFailed : BOOL;
    {attribute addProperty Name "<#Extended user data set acknowledge#>"}
    ExtendedUserDataSetAcknowledge : BOOL;
    {attribute addProperty Name "<#Overall job pass fail#>"}
    OverallJobPassFail : BOOL;
    {attribute addProperty Name "<#Test run ready#>"}
    TestRunReady : BOOL;
    {attribute addProperty Name "<#Error#>"}
    Error : BOOL;
    {attribute addProperty Name "<#Error code#>"}
    ErrorCode : UINT;
    {attribute wpf [Container(Layout.Stack,"Command control")]}
    {attribute wpf [Group(Layout.GroupBox)]}
    {attribute addProperty Name "<#Command#>"}
    Command : UINT;
    {attribute addProperty Name "<#Current job ID#>"}
    CurrentJobID : UINT;
    {attribute wpf [Container(Layout.Stack,"Command control")]}
    {attribute wpf [Group(Layout.GroupBox)]}
    {attribute addProperty Name "<#Trigger soft event#>"}
    TriggerSoftEvent : BYTE;
    {attribute addProperty Name "<#Trigger soft event acknowledge#>"}
    TriggerSoftEventAcknowledge : BYTE;
    {attribute wpf [Container(Layout.Stack,"Results data")]}
    {attribute wpf [Group(Layout.GroupBox)]}
    {attribute addProperty Name "<#Inspection ID#>"}
    InspectionID : UINT;
    {attribute addProperty Name "<#Result code#>"}
    ResultCode : UINT;
END_STRUCT
END_TYPE

// ---- POUs/TcoInsight/v_5_x_x/Structs/TcoInsightStatus_v_5_x_x.TcDUT
TYPE TcoInsightStatus_v_5_x_x :
STRUCT
    ActionDescription : STRING(100);
    SignalStatus : TcoInsightSignalStates_v_5_x_x;
    CurrentJobName : STRING(100);
    CurrentJobNumber : INT := -1;
END_STRUCT
END_TYPE

// ---- POUs/TcoInsight/v_5_x_x/Structs/TcoInsightUser_v_5_x_x.TcDUT
TYPE TcoInsightUser_v_5_x_x :
STRUCT
    UserData : ARRAY[0..TcoVisionParams.MAX_BYTE_ARRAY] OF BYTE;
END_STRUCT
END_TYPE

// ---- POUs/TcoVisionParams.TcGVL
{attribute 'qualified_only'}
VAR_GLOBAL CONSTANT
    MAX_BYTE_ARRAY : UINT := 255;
END_VAR

// ---- POUs/TcoDataman/v_5_x_x/Tasks/TcoDatamanClearResultData_v_5_x_x.TcPOU
FUNCTION_BLOCK TcoDatamanClearResultData_v_5_x_x EXTENDS TcoCore.TcoTask
VAR_IN_OUT
    inoIoData : TcoDatamanIO_v_5_x_x;
    inoConfig : TcoDatamanConfig_v_5_x_x;
    inoStatus : TcoDatamanStatus_v_5_x_x;
    inoResults : TcoDatamanResults_v_5_x_x;
END_VAR
VAR
    {attribute 'hide'}
    _progress : INT := 0;
    {attribute 'hide'}
    _infoTimer : TON;
    {attribute 'hide'}
    _errorTimer : TON;
    {attribute 'hide'}
    _varInfo : __SYSTEM.VAR_INFO;
    {attribute 'hide'}
    _sb : TcoCore.StringBuilder;
END_VAR

IF Execute() THEN
    IF _progress = 0 THEN
        IF NOT __ISVALIDREF(inoIoData) THEN
            _varInfo := __VARINFO(inoIoData);
            Messenger.Programming(_sb.Clear().Append('<#Invalid reference: #>').Append(_varInfo.Symbol).ToString()).Pin();
        ELSIF NOT __ISVALIDREF(inoConfig) THEN
            _varInfo := __VARINFO(inoConfig);
            Messenger.Programming(_sb.Clear().Append('<#Invalid reference: #>').Append(_varInfo.Symbol).ToString()).Pin();
        ELSIF NOT __ISVALIDREF(inoStatus) THEN
            _varInfo := __VARINFO(inoStatus);
            Messenger.Programming(_sb.Clear().Append('<#Invalid reference: #>').Append(_varInfo.Symbol).ToString()).Pin();
        ELSIF NOT __ISVALIDREF(inoResults) THEN
            _varInfo := __VARINFO(inoResults);
            Messenger.Programming(_sb.Clear().Append('<#Invalid reference: #>').Append(_varInfo.Symbol).ToString()).Pin();
        ELSE
            _progress := _progress + 1;
        END_IF
    END_IF

    IF _progress = 1 THEN
        THIS^.inoStatus.ActionDescription := '<#Clearing of the result data running.#>';
        CallTimers(FALSE);
        _progress := _progress + 1;
    END_IF

    IF _progress = 2 THEN
        THIS^.inoIoData.AcquisitionControl.TriggerEnable := FALSE;
        THIS^.inoIoData.AcquisitionControl.Trigger := FALSE;
        THIS^.inoIoData.ResultsControl.ResultsAcknowledge := TRUE;
        THIS^.Messenger.OnCondition(_infoTimer.Q).Warning('<#Waiting for the result data cleared!#>').Pin();
        THIS^.inoResults.Length := 0;

        IF Tc2_System.MEMSET(destAddr := ADR(THIS^.inoResults.Data), fillByte := 0, n := SIZEOF(THIS^.inoResults.Data)) > 0 THEN
            CallTimers(FALSE);
            _progress := _progress + 1;
        END_IF
    END_IF

    IF _progress = 3 THEN
        THIS^.Messenger.OnCondition(_infoTimer.Q).Warning('<#Waiting for the signal ResultsAvailable to be reseted!#>').Pin();

        IF NOT THIS^.inoIoData.ResultsStatus.ResultsAvailable THEN
            CallTimers(FALSE);
            _progress := _progress + 1;
        END_IF
    END_IF

    IF _progress = 4 THEN
        THIS^.inoIoData.ResultsControl.ResultsAcknowledge := FALSE;
        THIS^.DoneWhen(TRUE);
        CallTimers(FALSE);
        _progress := 0;
    END_IF

    CallTimers(TRUE);
    THIS^.ThrowWhen(_errorTimer.Q);
END_IF

METHOD CallTimers
VAR_INPUT
    inValue : BOOL;
END_VAR
_infoTimer(IN := inValue, PT := THIS^.inoConfig.InfoTime);
_errorTimer(IN := inValue, PT := THIS^.inoConfig.ErrorTime);
END_METHOD

{attribute 'hide'}
METHOD PUBLIC FB_init : BOOL
VAR_INPUT
    bInitRetains : BOOL; // if TRUE, the retain variables are initialized (warm start / cold start)
    bInCopyCode : BOOL; // if TRUE, the instance afterwards gets moved into the copy code (online change)
    ParentObject : ITcoObject;
END_VAR
END_METHOD

(*~
    <docu>
        <summary>
            Executes when task is aborted.
        </summary>
    </docu>
~*)
METHOD PROTECTED OnAbort
THIS^.inoStatus.ActionDescription := '<#Clearing of the result data was aborted, while not yet completed!#>';
END_METHOD

(*~
    <docu>
        <summary>
            Executes when task reaches the ```Done``` state .
        </summary>
    </docu>
~*)
METHOD PROTECTED OnDone
THIS^.inoStatus.ActionDescription := '<#Clearing of the result data was completed successfully.#>';
END_METHOD

(*~
    <docu>
        <summary>
            Executes when task reaches the ```Error``` state.
            <para>
                Do not confuse with <see cref="PlcDocu.TcoCore.TcoTask.WhileError()"/>, that is called cyclically until '''Error''' state is left.
            </para>
        </summary>
    </docu>
~*)
METHOD PROTECTED OnError
THIS^.inoStatus.ActionDescription := '<#Clearing of the result data finished with error.#>';
END_METHOD

METHOD PROTECTED OnStart
THIS^.inoStatus.ActionDescription := '<#Clearing of the result data started.#>';
END_METHOD

(*~
    <docu>
        <summary>
            Restores this instance to the Ready state. Can be called explicitly or from within one of the restore mechanisms.
            <para>
                See also <see cref="PlcDocu.TcoCore.TcoTask.AutoRestorable()"/>
            </para>
        </summary>
    </docu>
~*)
METHOD Restore : ITcoRestorable
SUPER^.Restore();
_progress := 0;
CallTimers(FALSE);
Messenger.UnPin();
END_METHOD

END_FUNCTION_BLOCK

// ---- POUs/TcoDataman/v_5_x_x/Tasks/TcoDatamanRead_v_5_x_x.TcPOU
FUNCTION_BLOCK TcoDatamanRead_v_5_x_x EXTENDS TcoCore.TcoTask
VAR_IN_OUT
    inoIoData : TcoDatamanIO_v_5_x_x;
    inoConfig : TcoDatamanConfig_v_5_x_x;
    inoStatus : TcoDatamanStatus_v_5_x_x;
    inoResults : TcoDatamanResults_v_5_x_x;
END_VAR
VAR
    {attribute 'hide'}
    _progress : INT := 0;
    {attribute 'hide'}
    _infoTimer : TON;
    {attribute 'hide'}
    _errorTimer : TON;
    {attribute 'hide'}
    _varInfo : __SYSTEM.VAR_INFO;
    {attribute 'hide'}
    _sb : TcoCore.StringBuilder;
END_VAR

IF Execute() THEN
    IF _progress = 0 THEN
        IF NOT __ISVALIDREF(inoIoData) THEN
            _varInfo := __VARINFO(inoIoData);
            Messenger.Programming(_sb.Clear().Append('<#Invalid reference: #>').Append(_varInfo.Symbol).ToString()).Pin();
        ELSIF NOT __ISVALIDREF(inoConfig) THEN
            _varInfo := __VARINFO(inoConfig);
            Messenger.Programming(_sb.Clear().Append('<#Invalid reference: #>').Append(_varInfo.Symbol).ToString()).Pin();
        ELSIF NOT __ISVALIDREF(inoStatus) THEN
            _varInfo := __VARINFO(inoStatus);
            Messenger.Programming(_sb.Clear().Append('<#Invalid reference: #>').Append(_varInfo.Symbol).ToString()).Pin();
        ELSIF NOT __ISVALIDREF(inoResults) THEN
            _varInfo := __VARINFO(inoResults);
            Messenger.Programming(_sb.Clear().Append('<#Invalid reference: #>').Append(_varInfo.Symbol).ToString()).Pin();
        ELSE
            _progress := _progress + 1;
        END_IF
    END_IF

    IF _progress = 1 THEN
        THIS^.inoStatus.ActionDescription := '<#Reading running.#>';
        CallTimers(FALSE);
        _progress := _progress + 1;
    END_IF

    IF _progress = 2 THEN
        THIS^.inoIoData.AcquisitionControl.TriggerEnable := TRUE;
        THIS^.inoIoData.AcquisitionControl.Trigger := FALSE;
        THIS^.inoIoData.ResultsControl.EnableResultBuffering := FALSE;
        THIS^.inoIoData.ResultsControl.ResultsAcknowledge := THIS^.inoIoData.ResultsStatus.ResultsAvailable;
        THIS^.Messenger.OnCondition(_infoTimer.Q).Warning('<#Waiting for the signal ResultsAvailable to be reseted!#>').Pin();

        IF NOT THIS^.inoIoData.ResultsStatus.ResultsAvailable THEN
            CallTimers(FALSE);
            _progress := _progress + 1;
        END_IF
    END_IF

    IF _progress = 3 THEN
        THIS^.Messenger.OnCondition(_infoTimer.Q).Warning('<#Waiting for the signal TriggerReady to be set!#>').Pin();

        IF THIS^.inoIoData.AcquisitionStatus.TriggerReady THEN
            CallTimers(FALSE);
            _progress := _progress + 1;
        END_IF
    END_IF

    IF _progress = 4 THEN
        THIS^.inoIoData.AcquisitionControl.Trigger := TRUE;
        THIS^.Messenger.OnCondition(_infoTimer.Q).Warning('<#Waiting for the signal TriggerAcknowledge to be set!#>').Pin();

        IF THIS^.inoIoData.AcquisitionStatus.TriggerAcknowledge THEN
            CallTimers(FALSE);
            _progress := _progress + 1;
        END_IF
    END_IF

    IF _progress = 5 THEN
        THIS^.Messenger.OnCondition(_infoTimer.Q).Warning('<#Waiting for the signal ResultsAvailable to be set!#>').Pin();

        IF THIS^.inoIoData.ResultsStatus.ResultsAvailable THEN
            CallTimers(FALSE);
            _progress := _progress + 1;
        END_IF
    END_IF

    IF _progress = 6 THEN
        THIS^.inoResults.Length := THIS^.inoIoData.ResultData.ResultLength;
        THIS^.Messenger.OnCondition(_infoTimer.Q).Warning('<#Waiting for the ResultData copied!#>').Pin();

        IF Tc2_System
            .MEMCPY(srcAddr := ADR(THIS^.inoIoData.ResultData.ResultData), destAddr := ADR(THIS^.inoResults.Data), n := THIS^.inoResults.Length) >
            0 AND
            Tc2_System.MEMSET(destAddr :=
                ADR(THIS^.inoResults.Data) + THIS^.inoResults.Length,
                fillByte := 0,
                n := SIZEOF(THIS^.inoResults.Data) - THIS^.inoResults.Length) >
            0 THEN
            CallTimers(FALSE);
            _progress := _progress + 1;
        END_IF
    END_IF

    IF _progress = 7 THEN
        THIS^.inoIoData.AcquisitionControl.Trigger := FALSE;
        THIS^.inoIoData.ResultsControl.EnableResultBuffering := FALSE;
        THIS^.inoIoData.ResultsControl.ResultsAcknowledge := TRUE;
        THIS^.ThrowWhen(THIS^.inoIoData.ResultData.ResultCode = 0 OR THIS^.inoIoData.ResultData.ResultLength = 0);
        THIS^.DoneWhen(TRUE);
        _progress := 0;
    END_IF

    CallTimers(TRUE);
    THIS^.ThrowWhen(_errorTimer.Q);
END_IF

METHOD CallTimers
VAR_INPUT
    inValue : BOOL;
END_VAR
_infoTimer(IN := inValue, PT := THIS^.inoConfig.InfoTime);
_errorTimer(IN := inValue, PT := THIS^.inoConfig.ErrorTime);
END_METHOD

{attribute 'hide'}
METHOD PUBLIC FB_init : BOOL
VAR_INPUT
    bInitRetains : BOOL; // if TRUE, the retain variables are initialized (warm start / cold start)
    bInCopyCode : BOOL; // if TRUE, the instance afterwards gets moved into the copy code (online change)
    ParentObject : ITcoObject;
END_VAR
END_METHOD

(*~
    <docu>
        <summary>
            Executes when task is aborted.
        </summary>
    </docu>
~*)
METHOD PROTECTED OnAbort
THIS^.inoStatus.ActionDescription := '<#Reading was aborted, while not yet completed!#>';
END_METHOD

(*~
    <docu>
        <summary>
            Executes when task reaches the ```Done``` state .
        </summary>
    </docu>
~*)
METHOD PROTECTED OnDone
THIS^.inoStatus.ActionDescription := '<#Reading was completed successfully.#>';
END_METHOD

(*~
    <docu>
        <summary>
            Executes when task reaches the ```Error``` state.
            <para>
                Do not confuse with <see cref="PlcDocu.TcoCore.TcoTask.WhileError()"/>, that is called cyclically until '''Error''' state is left.
            </para>
        </summary>
    </docu>
~*)
METHOD PROTECTED OnError
THIS^.inoStatus.ActionDescription := '<#Reading finished with error.#>';
END_METHOD

METHOD PROTECTED OnStart
THIS^.inoStatus.ActionDescription := '<#Reading started.#>';
THIS^.inoStatus.ResultString := '';
END_METHOD

(*~
    <docu>
        <summary>
            Restores this instance to the Ready state. Can be called explicitly or from within one of the restore mechanisms.
            <para>
                See also <see cref="PlcDocu.TcoCore.TcoTask.AutoRestorable()"/>
            </para>
        </summary>
    </docu>
~*)
METHOD Restore : ITcoRestorable
SUPER^.Restore();
_progress := 0;
CallTimers(FALSE);
Messenger.UnPin();
END_METHOD

END_FUNCTION_BLOCK

// ---- POUs/TcoDataman/v_5_x_x/TcoDataman_v_5_x_x.TcPOU
FUNCTION_BLOCK TcoDataman_v_5_x_x EXTENDS TcoIo.TcoPnIoComponent IMPLEMENTS TcoAbstractions.ITcoCodeReader
VAR_IN_OUT
    inoIoData : TcoDatamanIO_v_5_x_x;
END_VAR
VAR
    {attribute addProperty Name "<#Config#>"}
    _config : TcoDatamanConfig_v_5_x_x;
    {attribute addProperty Name "<#Status#>"}
    _status : TcoDatamanStatus_v_5_x_x;
END_VAR
VAR
    {attribute addProperty Name "<#UserData#>"}
    _userData : TcoDatamanUser_v_5_x_x;
    {attribute addProperty Name "<#Results#>"}
    _results : TcoDatamanResults_v_5_x_x;
END_VAR
VAR
    {attribute 'hide'}
    _taskEnabled : BOOL;
    {attribute addProperty Name "<#Restore#>"}
    _restoreTask : TcoCore.TcoTask(THIS^);
    {attribute addProperty Name "<#Update signal states#>"}
    _updateSignalStatesTask : TcoCore.TcoTask(THIS^);
    {attribute addProperty Name "<#Clear result data#>"}
    _clearResultDataTask : TcoDatamanClearResultData_v_5_x_x(THIS^);
    {attribute addProperty Name "<#Read#>"}
    _readTask : TcoDatamanRead_v_5_x_x(THIS^);
END_VAR
VAR
    {attribute 'hide'}
    _varInfo : __SYSTEM.VAR_INFO;
    {attribute 'hide'}
    _sb : TcoCore.StringBuilder;
END_VAR

IF InvalidReference() THEN
    RETURN;
END_IF

SUPER^(inPnIoBoxState := THIS^.inoIoData.PnIoBoxState, inPnIoBoxDiag := THIS^.inoIoData.PnIoBoxDiag);

IF THIS^._config.ContinuousReading THEN
    ContinuousReading();
END_IF

IF NOT SUPER^.ProfinetReady THEN
    THIS^._status.ActionDescription := '<#Not ready for operation by means of Profinet network!#>';
END_IF

IF SUPER^.ProfinetReady AND THIS^._status.ActionDescription = '<#Not ready for operation by means of Profinet network!#>' THEN
    THIS^._status.ActionDescription := '<#Ready for operation!#>';
END_IF
//*************RESTORE********************
_taskEnabled := TRUE;
_restoreTask.Enabled := _taskEnabled;

IF _restoreTask.Execute() THEN
    Restore();
END_IF

//****************************************
//*************UPDATE*********************
IF _config.UpdateStatesPermanently THEN
    UpdateSignalStates();
END_IF;

_taskEnabled := SUPER^.ProfinetReady;
_updateSignalStatesTask.Enabled := _taskEnabled AND NOT _config.UpdateStatesPermanently;

IF _updateSignalStatesTask.Execute() THEN
    UpdateSignalStates();
END_IF
//****************************************
//*************CLEAR*DATA*****************
_taskEnabled := SUPER^.ProfinetReady AND NOT _readTask.Busy;
_clearResultDataTask.Enabled := _taskEnabled;

_clearResultDataTask(inoIoData := THIS^.inoIoData,
    inoConfig := THIS^._config,
    inoStatus := THIS^._status,
    inoResults := THIS^._results);
//****************************************
//*************READ***********************
_taskEnabled := SUPER^.ProfinetReady AND NOT _clearResultDataTask.Busy;
_readTask.Enabled := _taskEnabled;

_readTask(inoIoData := THIS^.inoIoData,
    inoConfig := THIS^._config,
    inoStatus := THIS^._status,
    inoResults := THIS^._results);

IF NOT _readTask.Busy AND NOT _readTask.Error AND NOT _clearResultDataTask.Busy AND NOT _clearResultDataTask.Error THEN
    _status.ResultString := GetResultAsString(0, _status.SignalStatus.ResultLength);
END_IF;
//****************************************

(*~
    <docu>
        <summary>
            Clears the result data.
        </summary>
    </docu>
~*)
METHOD ClearResultData : TcoCore.ITcoTaskStatus
ClearResultData := THIS^._clearResultDataTask.Invoke();
END_METHOD

(*~
    <docu>
        <summary>
            Gets the `ClearResultDataTask` task that controls clearing of the results data.
        </summary>
    </docu>
~*)
PROPERTY ClearResultDataTask : TcoCore.ITcoTaskStatus
GET
ClearResultDataTask := _clearResultDataTask;
END_GET
END_PROPERTY

(*~
    <docu>
        <summary>
            Gets the configuration of the reader.
        </summary>
    </docu>
~*)
PROPERTY Config : REFERENCE TO TcoDatamanConfig_v_5_x_x
GET
Config REF= _config;
END_GET
END_PROPERTY

METHOD INTERNAL ContinuousReading
IF THIS^.inoIoData.ResultsStatus.ResultsAvailable AND
    NOT THIS^.inoIoData.ResultsControl.ResultsAcknowledge AND
    THIS^.inoIoData.ResultData.ResultCode > 0 AND
    THIS^.inoIoData.ResultData.ResultLength > 0 THEN
    THIS^._results.Length := THIS^.inoIoData.ResultData.ResultLength;
    Tc2_System.MEMCPY(srcAddr := ADR(THIS^.inoIoData.ResultData.ResultData), destAddr := ADR(THIS^._results.Data), n := THIS^._results.Length);

    Tc2_System.MEMSET(destAddr
            := ADR(THIS^._results.Data) + THIS^._results.Length,
        fillByte := 0,
        n := SIZEOF(THIS^._results.Data) - THIS^._results.Length);

    THIS^._status.ActionDescription := '<#New data read.#>';
END_IF

THIS^.inoIoData.ResultsControl.ResultsAcknowledge := THIS^.inoIoData.ResultsStatus.ResultsAvailable;
END_METHOD

METHOD FB_init : BOOL
VAR_INPUT
    bInitRetains : BOOL; // if TRUE, the retain variables are initialized (warm start / cold start)
    bInCopyCode : BOOL; // if TRUE, the instance afterwards gets moved into the copy code (online change)
    ParentObject : ITcoObject;
END_VAR
END_METHOD

METHOD GetResultAsByte : BYTE
VAR_INPUT
    inPosition : UINT;
END_VAR
VAR
    _size : UINT;
END_VAR
_size := SIZEOF(GetResultAsByte);

IF (inPosition + _size) > THIS^._results.Length THEN
    Messenger.Info('<#Index of the ResultData in the method GetResultAsByte exceeds the length of the data received!#>');
    RETURN;
END_IF

IF (inPosition + _size) > THIS^._config.ResultDataSize THEN
    Messenger.Warning('<#Index of the ResultData in the method GetResultAsByte exceeds the size hardware structure mapped!#>');
    RETURN;
END_IF

IF (inPosition + _size) > TcoVisionParams.MAX_BYTE_ARRAY THEN
    Messenger.Programming('<#Index of the ResultData in the method GetResultAsByte exceeds the defined size!#>');
    RETURN;
END_IF

GetResultAsByte := THIS^._results.Data[inPosition];
END_METHOD

METHOD GetResultAsDint : DINT
VAR_INPUT
    inPosition : UINT;
END_VAR
VAR
    _index : UINT;
    _size : UINT;
END_VAR
_size := SIZEOF(GetResultAsDint);

IF (inPosition + _size) > THIS^._results.Length THEN
    Messenger.Info('<#Index of the ResultData in the method GetResultAsDint exceeds the length of the data received!#>');
    RETURN;
END_IF

IF (inPosition + _size) > THIS^._config.ResultDataSize THEN
    Messenger.Warning('<#Index of the ResultData in the method GetResultAsDint exceeds the size hardware structure mapped!#>');
    RETURN;
END_IF

IF (inPosition + _size) > TcoVisionParams.MAX_BYTE_ARRAY THEN
    Messenger.Programming('<#Index of the ResultData in the method GetResultAsDint exceeds the defined size!#>');
    RETURN;
END_IF

GetResultAsDint := TcoUtilities.TcoBytesToDint(THIS^._config.DataFormat,
    THIS^._results.Data[inPosition],
    THIS^._results.Data[inPosition + 1],
    THIS^._results.Data[inPosition + 2],
    THIS^._results.Data[inPosition + 3]);
END_METHOD

METHOD GetResultAsReal : REAL
VAR_INPUT
    inPosition : UINT;
END_VAR
VAR
    _index : UINT;
    _size : UINT;
END_VAR
_size := SIZEOF(GetResultAsReal);

IF (inPosition + _size) > THIS^._results.Length THEN
    Messenger.Info('<#Index of the ResultData in the method GetResultAsReal exceeds the length of the data received!#>');
    RETURN;
END_IF

IF (inPosition + _size) > THIS^._config.ResultDataSize THEN
    Messenger.Warning('<#Index of the ResultData in the method GetResultAsReal exceeds the size hardware structure mapped!#>');
    RETURN;
END_IF

IF (inPosition + _size) > TcoVisionParams.MAX_BYTE_ARRAY THEN
    Messenger.Programming('<#Index of the ResultData in the method GetResultAsReal exceeds the defined size!#>');
    RETURN;
END_IF

GetResultAsReal := TcoUtilities.TcoBytesToReal(THIS^._config.DataFormat,
    THIS^._results.Data[inPosition],
    THIS^._results.Data[inPosition + 1],
    THIS^._results.Data[inPosition + 2],
    THIS^._results.Data[inPosition + 3]);
END_METHOD

METHOD GetResultAsString : STRING
VAR_INPUT
    inPosition : UINT;
    inLength : UINT;
END_VAR
VAR
    _index : UINT;
    _bufferSize : UINT;
    _resultString : STRING;
END_VAR
IF (inPosition + inLength) > THIS^._results.Length THEN
    Messenger.Info('<#Index of the ResultData in the method GetResultAsString exceeds the length of the data received!#>');
    RETURN;
END_IF

IF (inPosition + inLength) > THIS^._config.ResultDataSize THEN
    Messenger.Warning('<#Index of the ResultData in the method GetResultAsString exceeds the size hardware structure mapped!#>');
    RETURN;
END_IF

IF (inPosition + inLength) > TcoVisionParams.MAX_BYTE_ARRAY THEN
    Messenger.Programming('<#Index of the ResultData in the method GetResultAsString exceeds the defined size!#>');
    RETURN;
END_IF

_resultString := '';

IF (inLength > 0) THEN
    FOR _index := 0 TO inLength - 1 BY 1 DO
        IF (THIS^._results.Data[inPosition + _index] <> 0) THEN
            _resultString := CONCAT(_resultString, F_ToCHR(THIS^._results.Data[inPosition + _index]));
        ELSE
            EXIT;
        END_IF
    END_FOR;
END_IF

GetResultAsString := _resultString;
END_METHOD

METHOD INTERNAL InvalidReference : BOOL
InvalidReference := FALSE;

IF NOT __ISVALIDREF(inoIoData) THEN
    _varInfo := __VARINFO(inoIoData);
    Messenger.Error(_sb.Clear().Append('<#Invalid reference: #>').Append(_varInfo.Symbol).ToString());
    InvalidReference := TRUE;
END_IF
END_METHOD

(*~
    <docu>
        <summary>
            Gets the last results data.
        </summary>
    </docu>
~*)
PROPERTY LastResultData : TcoDatamanResults_v_5_x_x
GET
LastResultData := THIS^._results;
END_GET
END_PROPERTY

(*~
    <docu>
        <summary>
            Triggers the reading sequence and waits for results.
        </summary>
    </docu>
~*)
METHOD Read : TcoCore.ITcoTaskStatus
Read := THIS^._readTask.Invoke();
END_METHOD

(*~
    <docu>
        <summary>
            Gets the `ReadTask` task that controls the reading sequence.
        </summary>
    </docu>
~*)
PROPERTY ReadTask : TcoCore.ITcoTaskStatus
GET
ReadTask := _readTask;
END_GET
END_PROPERTY

(*~
    <docu>
        <summary>
            Restores this instance to the Ready state. Can be called explicitly or from within one of the restore mechanisms.
        </summary>
    </docu>
~*)
METHOD Restore : ITcoRestorable
_updateSignalStatesTask.Restore();
_clearResultDataTask.Restore();
_readTask.Restore();
Tc2_System.MEMSET(destAddr := ADR(THIS^._results.Data), fillByte := 0, n := SIZEOF(THIS^._results.Data));
THIS^.inoIoData.AcquisitionControl.TriggerEnable := FALSE;
THIS^.inoIoData.AcquisitionControl.Trigger := FALSE;
THIS^._results.Code := 0;
THIS^._results.Extended := 0;
THIS^._results.Id := 0;
THIS^._results.Length := 0;

IF InvalidReference() THEN
    RETURN;
END_IF

Tc2_System.MEMSET(destAddr := ADR(THIS^.inoIoData), fillByte := 0, n := SIZEOF(THIS^.inoIoData));
_status.ActionDescription := '<#Restore executed!#>';
_restoreTask.Restore();
END_METHOD

(*~
    <docu>
        <summary>
            Custom service (manual, maintenance) logic.
            This method must be implemented in derived class.
        </summary>
    </docu>
~*)
METHOD PROTECTED ServiceMode
END_METHOD

(*~
    <docu>
        <summary>
            Gets the status of the reader.
        </summary>
    </docu>
~*)
PROPERTY Status : REFERENCE TO TcoDatamanStatus_v_5_x_x
GET
Status REF= _status;
END_GET
END_PROPERTY

METHOD INTERNAL UpdateSignalStates
_status.SignalStatus.TriggerEnable := inoIoData.AcquisitionControl.TriggerEnable;
_status.SignalStatus.Trigger := inoIoData.AcquisitionControl.Trigger;
_status.SignalStatus.EnableResultBuffering := inoIoData.ResultsControl.EnableResultBuffering;
_status.SignalStatus.ResultsAcknowledge := inoIoData.ResultsControl.ResultsAcknowledge;
_status.SignalStatus.TriggerReady := inoIoData.AcquisitionStatus.TriggerReady;
_status.SignalStatus.TriggerAcknowledge := inoIoData.AcquisitionStatus.TriggerAcknowledge;
_status.SignalStatus.Acquiring := inoIoData.AcquisitionStatus.Acquiring;
_status.SignalStatus.MissedAcquisition := inoIoData.AcquisitionStatus.MissedAcquisition;
_status.SignalStatus.TriggerID := inoIoData.AcquisitionStatus.TriggerID;
_status.SignalStatus.Decoding := inoIoData.ResultsStatus.Decoding;
_status.SignalStatus.DecodeComplete := inoIoData.ResultsStatus.DecodeComplete;
_status.SignalStatus.ResultsBufferOverrun := inoIoData.ResultsStatus.ResultsBufferOverrun;
_status.SignalStatus.ResultsAvailable := inoIoData.ResultsStatus.ResultsAvailable;
_status.SignalStatus.ErrorDetected := inoIoData.ResultsStatus.ErrorDetected;
_status.SignalStatus.ResultID := inoIoData.ResultData.ResultID;
_status.SignalStatus.ResultCode := inoIoData.ResultData.ResultCode;
_status.SignalStatus.ResultExtended := inoIoData.ResultData.ResultExtended;
_status.SignalStatus.ResultLength := inoIoData.ResultData.ResultLength;
_updateSignalStatesTask.DoneWhen(TRUE);
END_METHOD

END_FUNCTION_BLOCK

// ---- POUs/TcoDesigner/Structs/TcoDesignerRootContainer.TcPOU
FUNCTION_BLOCK TcoDesignerRootContainer EXTENDS TcoCore.TcoObject
VAR_INPUT
END_VAR
VAR_OUTPUT
END_VAR
VAR
END_VAR

END_FUNCTION_BLOCK

// ---- POUs/TcoDesigner/Tasks/TcoDesignerTrigger_v_2_x_x.TcPOU
FUNCTION_BLOCK TcoDesignerTrigger_v_2_x_x EXTENDS TcoCore.TcoTask
VAR_INPUT
    inTriggerType : eTcoDesignerTriggerType;
    refClearResultsTask : REFERENCE TO TcoDesignerClearInspectionResults_v_2_x_x;
END_VAR
VAR
    _clearResultsTask : REFERENCE TO TcoDesignerClearInspectionResults_v_2_x_x;
END_VAR
VAR_IN_OUT
    inoIoData : TcoDesignerData_2_x_x;
    inoConfig : TcoDesignerConfig_v_2_x_x;
    inoStatus : TcoDesignerStatus_v_2_x_x;
    //inoResults	: TcoInsightResults_v_5_x_x;
END_VAR
VAR
    _progress : INT := 0;
    {attribute 'hide'}
    _infoTimer : TON;
    {attribute 'hide'}
    _errorTimer : TON;
    {attribute 'hide'}
    _varInfo : __SYSTEM.VAR_INFO;
    {attribute 'hide'}
    _sb : TcoCore.StringBuilder;
END_VAR

IF NOT __ISVALIDREF(refClearResultsTask) THEN
    Messenger.Post('<#Invalid reference ClearResultsTask>', TcoCore.eMessageCategory.ProgrammingError);
    RETURN;
END_IF

_clearResultsTask REF= refClearResultsTask;

IF Execute() THEN
    IF _progress = 0 THEN
        IF NOT __ISVALIDREF(inoIoData) THEN
            _varInfo := __VARINFO(inoIoData);
            Messenger.Programming(_sb.Clear().Append('<#Invalid reference: #>').Append(_varInfo.Symbol).ToString()).Pin();
        ELSIF NOT __ISVALIDREF(inoConfig) THEN
            _varInfo := __VARINFO(inoConfig);
            Messenger.Programming(_sb.Clear().Append('<#Invalid reference: #>').Append(_varInfo.Symbol).ToString()).Pin();
        ELSIF NOT __ISVALIDREF(inoStatus) THEN
            _varInfo := __VARINFO(inoStatus);
            Messenger.Programming(_sb.Clear().Append('<#Invalid reference: #>').Append(_varInfo.Symbol).ToString()).Pin();
        ELSIF inTriggerType = eTcoDesignerTriggerType.TriggerWithTimeout AND inoConfig.ErrorTime < inoConfig.TriggerTimemout THEN
            Messenger.Error(_sb.Clear().Append('<#Error time is lower than timeout. Please check config!#>').ToString()).Pin();
        ELSE
            _progress := _progress + 1;
            CallTimers(FALSE);
        END_IF
    END_IF

    IF _progress = 1 THEN
        IF inTriggerType = eTcoDesignerTriggerType.TriggerFast THEN
            _progress := _progress + 1;
        ELSIF inTriggerType = eTcoDesignerTriggerType.TriggerWithTimeout THEN
            inoIoData.PlcToPc.Timeout := TIME_TO_UINT(inoConfig.TriggerTimemout);

            IF _clearResultsTask.Invoke().Done THEN
                _progress := _progress + 1;
            END_IF;
        ELSIF _clearResultsTask.Invoke().Done THEN
            _progress := _progress + 1;
        END_IF
    END_IF;

    IF _progress = 2 THEN
        THIS^.Messenger.OnCondition(_infoTimer.Q).Info('<#Trigger!#>');
        THIS^.inoIoData.PlcToPc.Trigger := TRUE;

        IF NOT THIS^.inoIoData.PcToPlc.InspectionReady THEN
            THIS^.inoIoData.PlcToPc.Trigger := FALSE;
            CallTimers(FALSE);
            _progress := _progress + 1;
        END_IF
    END_IF

    IF _progress = 3 THEN
        Messenger.Info('Waiting for results available');

        IF THIS^.inoIoData.PcToPlc.ResultsAvailable THEN
            CallTimers(FALSE);
            _progress := _progress + 1;
        END_IF
    END_IF

    IF _progress = 4 THEN
        Messenger.Info('Acknovledge results');
        THIS^.inoIoData.PlcToPc.ResultsAck := TRUE;

        IF NOT THIS^.inoIoData.PcToPlc.ResultsAvailable THEN
            THIS^.inoIoData.PlcToPc.ResultsAck := FALSE;
            THIS^.DoneWhen(TRUE);
        END_IF
    END_IF

    CallTimers(TRUE);

    THIS^.ThrowWhen(_errorTimer.Q OR
            THIS^.inoIoData.PcToPlc.Error OR
            (inTriggerType = eTcoDesignerTriggerType.TriggerWithTimeout AND THIS^.inoIoData.PcToPlc.TriggerTimeout));
END_IF

METHOD CallTimers
VAR_INPUT
    inValue : BOOL;
END_VAR
_infoTimer(IN := inValue, PT := THIS^.inoConfig.InfoTime);
_errorTimer(IN := inValue, PT := THIS^.inoConfig.ErrorTime);
END_METHOD

(*~
    <docu>
        <summary>
            Executes when task is aborted.
        </summary>
    </docu>
~*)
METHOD PROTECTED OnAbort
THIS^.inoStatus.ActionDescription := '<#Trigger was aborted, while not yet completed!#>';
END_METHOD

(*~
    <docu>
        <summary>
            Executes when task reaches the ```Done``` state .
        </summary>
    </docu>
~*)
METHOD PROTECTED OnDone
THIS^.inoStatus.ActionDescription := '<#Trigger was completed successfully.#>';
_progress := 0;
END_METHOD

(*~
    <docu>
        <summary>
            Executes when task reaches the ```Error``` state.
            <para>
                Do not confuse with <see cref="PlcDocu.TcoCore.TcoTask.WhileError()"/>, that is called cyclically until '''Error''' state is left.
            </para>
        </summary>
    </docu>
~*)
METHOD PROTECTED OnError
THIS^.inoStatus.ActionDescription := '<#Trigger finished with error.#>';
END_METHOD

METHOD PROTECTED OnStart
THIS^.inoStatus.ActionDescription := '<#Trigger started.#>';
inoIoData.PlcToPc.Timeout := 0;
END_METHOD

(*~
    <docu>
        <summary>
            Restores this instance to the Ready state. Can be called explicitly or from within one of the restore mechanisms.
            <para>
                See also <see cref="PlcDocu.TcoCore.TcoTask.AutoRestorable()"/>
            </para>
        </summary>
    </docu>
~*)
METHOD Restore : ITcoRestorable
SUPER^.Restore();
_progress := 0;
CallTimers(FALSE);
Messenger.UnPin();
END_METHOD

END_FUNCTION_BLOCK

// ---- POUs/TcoDesigner/Tasks/TcoDesignerClearInspectionResults_v_2_x_x.TcPOU
FUNCTION_BLOCK TcoDesignerClearInspectionResults_v_2_x_x EXTENDS TcoCore.TcoTask
VAR_IN_OUT
    inoIoData : TcoDesignerData_2_x_x;
    inoConfig : TcoDesignerConfig_v_2_x_x;
    inoStatus : TcoDesignerStatus_v_2_x_x;
    //inoResults	: TcoInsightResults_v_5_x_x;
END_VAR
VAR
    {attribute 'hide'}
    _progress : INT := 0;
    {attribute 'hide'}
    _infoTimer : TON;
    {attribute 'hide'}
    _errorTimer : TON;
    {attribute 'hide'}
    _varInfo : __SYSTEM.VAR_INFO;
    {attribute 'hide'}
    _sb : TcoCore.StringBuilder;
END_VAR

IF Execute() THEN
    IF _progress = 0 THEN
        IF NOT __ISVALIDREF(inoIoData) THEN
            _varInfo := __VARINFO(inoIoData);
            Messenger.Programming(_sb.Clear().Append('<#Invalid reference: #>').Append(_varInfo.Symbol).ToString()).Pin();
        ELSIF NOT __ISVALIDREF(inoConfig) THEN
            _varInfo := __VARINFO(inoConfig);
            Messenger.Programming(_sb.Clear().Append('<#Invalid reference: #>').Append(_varInfo.Symbol).ToString()).Pin();
        ELSIF NOT __ISVALIDREF(inoStatus) THEN
            _varInfo := __VARINFO(inoStatus);
            Messenger.Programming(_sb.Clear().Append('<#Invalid reference: #>').Append(_varInfo.Symbol).ToString()).Pin();
            //		ELSIF NOT __ISVALIDREF(inoResults) THEN
            //			_varInfo :=__VARINFO(inoResults);
        //			Messenger.Programming(_sb.Clear().Append('<#Invalid reference: #>').Append(_varInfo.Symbol).ToString()).Pin();
        ELSE
            _progress := _progress + 1;
        END_IF
    END_IF

    IF _progress = 1 THEN
        CallTimers(FALSE);
        THIS^.inoIoData.PlcToPc.Trigger := FALSE;
        THIS^.inoIoData.PlcToPc.LoadJob := FALSE;
        THIS^.inoIoData.PlcToPc.Reset := FALSE;
        THIS^.inoIoData.PlcToPc.ResultsAck := FALSE;
        THIS^.inoIoData.PlcToPc.ClearResults := FALSE;
        _progress := _progress + 1;
    END_IF

    IF _progress = 2 THEN
        THIS^.Messenger.OnCondition(_infoTimer.Q).Info('<#Reset Request!#>');
        THIS^.inoIoData.PlcToPc.Reset := TRUE;

        IF THIS^.inoIoData.PcToPlc.InspectionReady AND
            NOT THIS^.inoIoData.PcToPlc.ClearResultsAck AND
            NOT THIS^.inoIoData.PcToPlc.ResultsAvailable AND
            NOT THIS^.inoIoData.PcToPlc.JobLoadDone THEN
            THIS^.inoIoData.PlcToPc.Reset := FALSE;
            _progress := _progress + 1;
        END_IF
    END_IF

    IF _progress = 3 THEN
        THIS^.Messenger.OnCondition(_infoTimer.Q).Warning('<#Waiting for the Online signal!#>');

        IF THIS^.inoIoData.PcToPlc.SystemOnline THEN
            CallTimers(FALSE);
            _progress := _progress + 1;
        END_IF
    END_IF

    IF _progress = 4 THEN
        THIS^.Messenger.OnCondition(_infoTimer.Q).Info('<#Waiting to Acknowledge results!#>');
        THIS^.inoIoData.PlcToPc.ResultsAck := TRUE;

        IF NOT THIS^.inoIoData.PcToPlc.ResultsAvailable THEN
            THIS^.inoIoData.PlcToPc.ResultsAck := FALSE;
            CallTimers(FALSE);
            _progress := _progress + 1;
        END_IF
    END_IF

    IF _progress = 5 THEN
        THIS^.Messenger.OnCondition(_infoTimer.Q).Info('<#Waiting to clear old data!#>');
        THIS^.inoIoData.PlcToPc.ClearResults := TRUE;

        IF THIS^.inoIoData.PcToPlc.ClearResultsAck THEN
            THIS^.inoIoData.PlcToPc.ClearResults := FALSE;
            CallTimers(FALSE);
            _progress := _progress + 1;
        END_IF
    END_IF

    IF _progress = 6 THEN
        THIS^.Messenger.OnCondition(_infoTimer.Q).Info('<#Waiting for Inspection ready!#>');

        IF THIS^.inoIoData.PcToPlc.InspectionReady THEN
            CallTimers(FALSE);
            _progress := _progress + 1;
        END_IF
    END_IF

    IF _progress = 7 THEN
        THIS^.Messenger.OnCondition(_infoTimer.Q).Info('<#Waiting for data were cleared!#>');

        IF NOT THIS^.inoIoData.PcToPlc.ClearResultsAck AND
            NOT THIS^.inoIoData.PcToPlc.InspectionResults.ResultFail AND
            NOT THIS^.inoIoData.PcToPlc.InspectionResults.ResultPass THEN
            CallTimers(FALSE);
            THIS^.DoneWhen(TRUE);
        END_IF
    END_IF

    CallTimers(TRUE);
    THIS^.ThrowWhen(_errorTimer.Q OR THIS^.inoIoData.PcToPlc.Error);
END_IF

METHOD CallTimers
VAR_INPUT
    inValue : BOOL;
END_VAR
_infoTimer(IN := inValue, PT := THIS^.inoConfig.InfoTime);
_errorTimer(IN := inValue, PT := THIS^.inoConfig.ErrorTime);
END_METHOD

(*~
    <docu>
        <summary>
            Executes when task is aborted.
        </summary>
    </docu>
~*)
METHOD PROTECTED OnAbort
THIS^.inoStatus.ActionDescription := '<#Clearing of the inspection results aborted, while not yet finished.#>';
END_METHOD

(*~
    <docu>
        <summary>
            Executes when task reaches the ```Done``` state .
        </summary>
    </docu>
~*)
METHOD PROTECTED OnDone
THIS^.inoStatus.ActionDescription := '<#Clearing of the inspection results was completed succesfully.#>';
_progress := 0;
END_METHOD

(*~
    <docu>
        <summary>
            Executes when task reaches the ```Error``` state.
            <para>
                Do not confuse with <see cref="PlcDocu.TcoCore.TcoTask.WhileError()"/>, that is called cyclically until '''Error''' state is left.
            </para>
        </summary>
    </docu>
~*)
METHOD PROTECTED OnError
THIS^.inoStatus.ActionDescription := '<#Clearing of the inspection results finished with error.#>';
END_METHOD

METHOD PROTECTED OnStart
THIS^.inoStatus.ActionDescription := '<#Clearing of the inspection results started.#>';
END_METHOD

(*~
    <docu>
        <summary>
            Restores this instance to the Ready state. Can be called explicitly or from within one of the restore mechanisms.
            <para>
                See also <see cref="PlcDocu.TcoCore.TcoTask.AutoRestorable()"/>
            </para>
        </summary>
    </docu>
~*)
METHOD Restore : ITcoRestorable
SUPER^.Restore();
_progress := 0;
CallTimers(FALSE);
Messenger.UnPin();
END_METHOD

END_FUNCTION_BLOCK

// ---- POUs/TcoDesigner/TcoDesigner_v_2_x_x.TcPOU
FUNCTION_BLOCK TcoDesigner_v_2_x_x EXTENDS TcoCore.TcoComponent
VAR_IN_OUT
    inoData : TcoDesignerRootContainer;
END_VAR
VAR
    {attribute addProperty Name "<#Generic Data#>"}
    _genericData : TcoDesignerData_2_x_x;
    {attribute addProperty Name "<#Config#>"}
    _config : TcoDesignerConfig_v_2_x_x;
    {attribute addProperty Name "<#Status#>"}
    _status : TcoDesignerStatus_v_2_x_x;
    _triggerType : eTcoDesignerTriggerType;
    _internalLiveBit : BOOL;
END_VAR
VAR
    {attribute 'hide'}
    _taskEnabled : BOOL;
    {attribute addProperty Name "<#Restore#>"}
    _restoreTask : TcoCore.TcoTask(THIS^);
    {attribute addProperty Name "<#Clear result data#>"}
    _clearResultDataTask : TcoDesignerClearInspectionResults_v_2_x_x(THIS^);
    {attribute clr [RenderIgnore()]}
    _triggerInternalTask : TcoDesignerTrigger_v_2_x_x(THIS^);
    {attribute addProperty Name "<#Trigger#>"}
    _triggerTask : TcoCore.TcoTask(THIS^);
    {attribute addProperty Name "<#Trigger Fast#>"}
    _triggerFastTask : TcoCore.TcoTask(THIS^);
    {attribute addProperty Name "<#Trigger with Timeout#>"}
    _triggerWithTimeoutTask : TcoCore.TcoTask(THIS^);
    {attribute addProperty Name "<#Results#>"}
    {attribute clr [MemberByIdentity()]}
    _specificData : TcoDesignerRootContainer(THIS^);
    _timerConnection : TON;
END_VAR
VAR
    {attribute 'hide'}
    _varInfo : __SYSTEM.VAR_INFO;
    {attribute 'hide'}
    _sb : TcoCore.StringBuilder;
END_VAR

_specificData := inoData;
_status.SignalStatus := _genericData.PcToPlc;
_timerConnection(In := _internalLiveBit XOR _status.SignalStatus.LiveBit, PT := _config.ConnectionTimemout);
_status.ClientConnected := NOT _timerConnection.Q; //_timerConnection.ET<_timerConnection.PT AND _timerConnection.ET<>T#0MS;
_internalLiveBit := NOT _status.SignalStatus.LiveBit;

IF NOT _status.ClientConnected THEN
    THIS^._status.ActionDescription := '<#Vision system is not  responding via Ads. Check connection with Cognex Designer!#>';
    THIS^.Messenger.Error(_status.ActionDescription).Pin();
END_IF
//*************RESTORE********************
_restoreTask.Enabled := TRUE;

IF _restoreTask.Execute() THEN
    Restore();
    _restoreTask.DoneWhen(TRUE);
END_IF
//****************************************
//****************************************
//*************CLEAR*DATA*****************
_clearResultDataTask.Enabled := _status.ClientConnected;
_clearResultDataTask(inoIoData := _genericData, inoConfig := THIS^._config, inoStatus := THIS^._status);
//****************************************
//*************TRIGGER ********************
_triggerTask.Enabled := NOT _triggerFastTask.Busy AND NOT _triggerWithTimeoutTask.Busy AND _status.ClientConnected;

IF _triggerTask.Execute() THEN
    _triggerInternalTask.Enabled := TRUE;
    _triggerType := eTcoDesignerTriggerType.Trigger;
    _triggerTask.DoneWhen(_triggerInternalTask.Invoke().Done);
    _triggerTask.ThrowWhen(_triggerInternalTask.Error);
END_IF
//***********************************************
//*************TRIGGER WITH TIMEOUT********************
_triggerWithTimeoutTask.Enabled := NOT _triggerFastTask.Busy AND NOT _triggerTask.Busy AND _status.ClientConnected;

IF _triggerWithTimeoutTask.Execute() THEN
    _triggerInternalTask.Enabled := TRUE;
    _triggerType := eTcoDesignerTriggerType.TriggerWithTimeout;
    _triggerWithTimeoutTask.DoneWhen(_triggerInternalTask.Invoke().Done);
    _triggerWithTimeoutTask.ThrowWhen(_triggerInternalTask.Error);
END_IF
//***********************************************
//*************TRIGGER FAST********************
_triggerFastTask.Enabled := NOT _triggerWithTimeoutTask.Busy AND NOT _triggerTask.Busy AND _status.ClientConnected;

IF _triggerFastTask.Execute() THEN
    _triggerInternalTask.Enabled := TRUE;
    _triggerType := eTcoDesignerTriggerType.TriggerFast;
    _triggerFastTask.DoneWhen(_triggerInternalTask.Invoke().Done);
    _triggerFastTask.ThrowWhen(_triggerInternalTask.Error);
END_IF

//***********************************************
_triggerInternalTask(inTriggerType := _triggerType,
    refClearResultsTask := _clearResultDataTask,
    inoIoData := _genericData,
    inoConfig := THIS^._config,
    inoStatus := THIS^._status);

inoData := _specificData;

(*~
    <docu>
        <summary>
            Clears the result data.
        </summary>
    </docu>
~*)
METHOD ClearResultData : TcoCore.ITcoTaskStatus
ClearResultData := THIS^._clearResultDataTask.Invoke();
END_METHOD

(*~
    <docu>
        <summary>
            Gets the `ClearResultDataTask` task that controls clearing of the results data.
        </summary>
    </docu>
~*)
PROPERTY ClearResultDataTask : TcoCore.ITcoTaskStatus
GET
ClearResultDataTask := _clearResultDataTask;
END_GET
END_PROPERTY

(*~
    <docu>
        <summary>
            Gets the status of ads connection
        </summary>
    </docu>
~*)
PROPERTY ClientConnected : BOOL
GET
ClientConnected := THIS^.Status.ClientConnected;
END_GET
END_PROPERTY

(*~
    <docu>
        <summary>
            Gets the configuration of the cognex designer.
        </summary>
    </docu>
~*)
PROPERTY Config : REFERENCE TO TcoDesignerConfig_v_2_x_x
GET
Config REF= _config;
END_GET
END_PROPERTY

(*~
    <docu>
        <summary>
            Restores this instance to the Ready state. Can be called explicitly or from within one of the restore mechanisms.
        </summary>
    </docu>
~*)
METHOD Restore : ITcoRestorable
_clearResultDataTask.Restore();
_triggerInternalTask.Restore();
_triggerTask.Restore();
_triggerFastTask.Restore();
_triggerWithTimeoutTask.Restore();
THIS^.Messenger.UnPin();
//Tc2_System.MEMSET(destAddr:= ADR(THIS^._results.Data) , fillByte:= 0 , n:= SIZEOF(THIS^._results.Data));
_genericData.PlcToPc.Trigger := FALSE;
_genericData.PlcToPc.LoadJob := FALSE;
_genericData.PlcToPc.ClearResults := FALSE;
_genericData.PlcToPc.Reset := FALSE;
_genericData.PlcToPc.ResultsAck := FALSE;
_genericData.PlcToPc.JobLoadId := 0;
_genericData.PlcToPc.PartId := '';
//Tc2_System.MEMSET(destAddr:= ADR(THIS^.inoIoData) , fillByte:= 0 , n:= SIZEOF(THIS^.inoIoData));
_status.ActionDescription := '<#Restore executed!#>';
END_METHOD

(*~
    <docu>
        <summary>
            Custom service (manual, maintenance) logic.
            This method must be implemented in derived class.
        </summary>
    </docu>
~*)
METHOD PROTECTED ServiceMode
END_METHOD

(*~
    <docu>
        <summary>
            Gets the status of the cognex designer.
        </summary>
    </docu>
~*)
PROPERTY Status : REFERENCE TO TcoDesignerStatus_v_2_x_x
GET
Status REF= _status;
END_GET
END_PROPERTY

(*~
    <docu>
        <summary>
            Triggers the designer  sequence and waits for results.
        </summary>
    </docu>
~*)
METHOD Trigger : TcoCore.ITcoTaskStatus
Trigger := THIS^._triggerInternalTask.Invoke();
END_METHOD

(*~
    <docu>
        <summary>
            Gets the `ReadTask` task that controls the reading sequence.
        </summary>
    </docu>
~*)
PROPERTY TriggerTask : TcoCore.ITcoTaskStatus
GET
TriggerTask := _triggerInternalTask;
END_GET
END_PROPERTY

END_FUNCTION_BLOCK

// ---- POUs/TcoInsight/v_5_x_x/Tasks/TcoInsightTrigger_v_5_x_x.TcPOU
FUNCTION_BLOCK TcoInsightTrigger_v_5_x_x EXTENDS TcoCore.TcoTask
VAR_IN_OUT
    inoIoData : TcoInsightIO_v_5_x_x;
    inoConfig : TcoInsightConfig_v_5_x_x;
    inoStatus : TcoInsightStatus_v_5_x_x;
    inoResults : TcoInsightResults_v_5_x_x;
END_VAR
VAR
    {attribute 'hide'}
    _progress : INT := 0;
    {attribute 'hide'}
    _infoTimer : TON;
    {attribute 'hide'}
    _errorTimer : TON;
    {attribute 'hide'}
    _varInfo : __SYSTEM.VAR_INFO;
    {attribute 'hide'}
    _sb : TcoCore.StringBuilder;
    {attribute 'hide'}
    _inspectionCompleted : BOOL;
    {attribute 'hide'}
    _size : UINT;
END_VAR

IF Execute() THEN
    IF _progress = 0 THEN
        IF NOT __ISVALIDREF(inoIoData) THEN
            _varInfo := __VARINFO(inoIoData);
            Messenger.Programming(_sb.Clear().Append('<#Invalid reference: #>').Append(_varInfo.Symbol).ToString()).Pin();
        ELSIF NOT __ISVALIDREF(inoConfig) THEN
            _varInfo := __VARINFO(inoConfig);
            Messenger.Programming(_sb.Clear().Append('<#Invalid reference: #>').Append(_varInfo.Symbol).ToString()).Pin();
        ELSIF NOT __ISVALIDREF(inoStatus) THEN
            _varInfo := __VARINFO(inoStatus);
            Messenger.Programming(_sb.Clear().Append('<#Invalid reference: #>').Append(_varInfo.Symbol).ToString()).Pin();
        ELSIF NOT __ISVALIDREF(inoResults) THEN
            _varInfo := __VARINFO(inoResults);
            Messenger.Programming(_sb.Clear().Append('<#Invalid reference: #>').Append(_varInfo.Symbol).ToString()).Pin();
        ELSE
            _progress := _progress + 1;
        END_IF
    END_IF

    IF _progress = 1 THEN
        THIS^.inoStatus.ActionDescription := '<#Trigger running.#>';
        CallTimers(FALSE);
        THIS^.inoIoData.AcquisitionControl.AcquisitionTriggerEnable := TRUE;
        THIS^.inoIoData.AcquisitionControl.AcquisitionTrigger := FALSE;
        THIS^.inoIoData.AcquisitionControl.ClearExposureComplete := THIS^.inoIoData.AcquisitionStatus.ExposureComplete;
        THIS^.inoIoData.AcquisitionControl.SetOffline := FALSE;
        THIS^.inoIoData.InspectionControl.EnableResultsBuffering := FALSE;
        THIS^.inoIoData.InspectionControl.AcknowledgeInspectionResults := THIS^.inoIoData.InspectionStatus.ResultsValid;
        THIS^.inoIoData.InspectionControl.ExtendedUserDataSet := FALSE;
        THIS^.inoIoData.InspectionControl.ExecuteCommand := FALSE;
        THIS^.inoIoData.InspectionControl.ClearError := THIS^.inoIoData.InspectionStatus.Error;
        THIS^.inoIoData.CommandControl.Command := 0;
        _progress := _progress + 1;
    END_IF

    IF _progress = 2 THEN
        THIS^.Messenger.OnCondition(_infoTimer.Q).Warning('<#Waiting for the signal ExposureComplete to be reseted!#>').Pin();

        IF NOT THIS^.inoIoData.AcquisitionStatus.ExposureComplete THEN
            THIS^.inoIoData.AcquisitionControl.ClearExposureComplete := FALSE;
            CallTimers(FALSE);
            _progress := _progress + 1;
        END_IF
    END_IF

    IF _progress = 3 THEN
        THIS^.Messenger.OnCondition(_infoTimer.Q).Warning('<#Waiting for the signal ResultsValid to be reseted!#>').Pin();

        IF NOT THIS^.inoIoData.InspectionStatus.ResultsValid THEN
            THIS^.inoIoData.InspectionControl.AcknowledgeInspectionResults := FALSE;
            CallTimers(FALSE);
            _progress := _progress + 1;
        END_IF
    END_IF

    IF _progress = 4 THEN
        THIS^.Messenger.OnCondition(_infoTimer.Q).Warning('<#Waiting for the signal Error to be reseted!#>').Pin();

        IF NOT THIS^.inoIoData.InspectionStatus.Error THEN
            THIS^.inoIoData.InspectionControl.ClearError := FALSE;
            CallTimers(FALSE);
            _progress := _progress + 1;
        END_IF
    END_IF

    IF _progress = 5 THEN
        THIS^.Messenger.OnCondition(_infoTimer.Q).Warning('<#Waiting for the signal AcquisitionTriggerReady to be set!#>').Pin();
        _inspectionCompleted := THIS^.inoIoData.InspectionStatus.InspectionCompleted;

        IF THIS^.inoIoData.AcquisitionStatus.AcquisitionTriggerReady THEN
            CallTimers(FALSE);
            _progress := _progress + 1;
        END_IF
    END_IF

    IF _progress = 6 THEN
        THIS^.Messenger.OnCondition(_infoTimer.Q).Warning('<#Waiting for the signal AcquisitionTriggerAcknowledge to be set!#>').Pin();
        THIS^.inoIoData.AcquisitionControl.AcquisitionTrigger := TRUE;

        IF THIS^.inoIoData.AcquisitionStatus.AcquisitionTriggerAcknowledge THEN
            CallTimers(FALSE);
            _progress := _progress + 1;
        END_IF
    END_IF

    IF _progress = 7 THEN
        THIS^.Messenger.OnCondition(_infoTimer.Q).Warning('<#Waiting for the signal InspectionCompleted to be toggled!#>').Pin();
        THIS^.inoIoData.AcquisitionControl.AcquisitionTrigger := FALSE;

        IF THIS^._inspectionCompleted <> THIS^.inoIoData.InspectionStatus.InspectionCompleted THEN
            CallTimers(FALSE);
            _progress := _progress + 1;
        END_IF
    END_IF

    IF _progress = 8 THEN
        THIS^.Messenger.OnCondition(_infoTimer.Q).Warning('<#Waiting for the signal ResultsValid to be set!#>').Pin();

        IF THIS^.inoIoData.InspectionStatus.ResultsValid THEN
            CallTimers(FALSE);
            _progress := _progress + 1;
        END_IF
    END_IF

    IF _progress = 9 THEN
        THIS^.Messenger.OnCondition(_infoTimer.Q).Warning('<#Waiting for the InspectionResults to be copied!#>').Pin();
        THIS^.inoResults.InspectionId := THIS^.inoIoData.ResultsData.InspectionID;
        THIS^.inoResults.ResultCode := THIS^.inoIoData.ResultsData.ResultCode;
        _size := THIS^.inoConfig.ResultDataSize;

        IF Tc2_System
            .MEMCPY(srcAddr := ADR(THIS^.inoIoData.ResultsData.InspectionResults), destAddr := ADR(THIS^.inoResults.InspectionResults), n := _size) >
            0 AND
            Tc2_System.MEMSET(destAddr := ADR(THIS^.inoResults.InspectionResults) + _size,
                fillByte := 0,
                n := SIZEOF(THIS^.inoResults.InspectionResults) - _size) >
            0 THEN
            CallTimers(FALSE);
            _progress := _progress + 1;
        END_IF
    END_IF

    IF _progress = 10 THEN
        THIS^.inoIoData.AcquisitionControl.AcquisitionTrigger := FALSE;
        THIS^.inoIoData.InspectionControl.EnableResultsBuffering := FALSE;
        THIS^.inoIoData.InspectionControl.AcknowledgeInspectionResults := TRUE;
        THIS^.ThrowWhen(THIS^.inoIoData.InspectionStatus.Error);
        THIS^.DoneWhen(TRUE);
        _progress := 0;
    END_IF

    CallTimers(TRUE);
    THIS^.ThrowWhen(_errorTimer.Q OR _progress > 4 AND THIS^.inoIoData.InspectionStatus.Error);
END_IF

METHOD CallTimers
VAR_INPUT
    inValue : BOOL;
END_VAR
_infoTimer(IN := inValue, PT := THIS^.inoConfig.InfoTime);
_errorTimer(IN := inValue, PT := THIS^.inoConfig.ErrorTime);
END_METHOD

{attribute 'hide'}
METHOD PUBLIC FB_init : BOOL
VAR_INPUT
    bInitRetains : BOOL; // if TRUE, the retain variables are initialized (warm start / cold start)
    bInCopyCode : BOOL; // if TRUE, the instance afterwards gets moved into the copy code (online change)
    ParentObject : ITcoObject;
END_VAR
END_METHOD

(*~
    <docu>
        <summary>
            Executes when task is aborted.
        </summary>
    </docu>
~*)
METHOD PROTECTED OnAbort
THIS^.inoStatus.ActionDescription := '<#Trigger was aborted, while not yet completed!#>';
END_METHOD

(*~
    <docu>
        <summary>
            Executes when task reaches the ```Done``` state .
        </summary>
    </docu>
~*)
METHOD PROTECTED OnDone
THIS^.inoStatus.ActionDescription := '<#Trigger was completed successfully.#>';
END_METHOD

(*~
    <docu>
        <summary>
            Executes when task reaches the ```Error``` state.
            <para>
                Do not confuse with <see cref="PlcDocu.TcoCore.TcoTask.WhileError()"/>, that is called cyclically until '''Error''' state is left.
            </para>
        </summary>
    </docu>
~*)
METHOD PROTECTED OnError
THIS^.inoStatus.ActionDescription := '<#Trigger finished with error.#>';
END_METHOD

METHOD PROTECTED OnStart
THIS^.inoStatus.ActionDescription := '<#Trigger started.#>';
END_METHOD

(*~
    <docu>
        <summary>
            Restores this instance to the Ready state. Can be called explicitly or from within one of the restore mechanisms.
            <para>
                See also <see cref="PlcDocu.TcoCore.TcoTask.AutoRestorable()"/>
            </para>
        </summary>
    </docu>
~*)
METHOD Restore : ITcoRestorable
SUPER^.Restore();
_progress := 0;
CallTimers(FALSE);
Messenger.UnPin();
END_METHOD

END_FUNCTION_BLOCK

// ---- POUs/TcoInsight/v_5_x_x/Tasks/TcoInsightChangeJobByName_v_5_x_x.TcPOU
FUNCTION_BLOCK TcoInsightChangeJobByName_v_5_x_x EXTENDS TcoCore.TcoTask
VAR_IN_OUT
    inoIoData : TcoInsightIO_v_5_x_x;
    inoConfig : TcoInsightConfig_v_5_x_x;
    inoStatus : TcoInsightStatus_v_5_x_x;
END_VAR
VAR
    {attribute addProperty Name "<#Job name#>"}
    _jobName : STRING;
END_VAR
VAR
    {attribute 'hide'}
    _progress : INT := 0;
    {attribute 'hide'}
    _infoTimer : TON;
    {attribute 'hide'}
    _errorTimer : TON;
    {attribute 'hide'}
    _varInfo : __SYSTEM.VAR_INFO;
    {attribute 'hide'}
    _sb : TcoCore.StringBuilder;
END_VAR

IF Execute() THEN
    IF _progress = 0 THEN
        IF NOT __ISVALIDREF(inoIoData) THEN
            _varInfo := __VARINFO(inoIoData);
            Messenger.Programming(_sb.Clear().Append('<#Invalid reference: #>').Append(_varInfo.Symbol).ToString()).Pin();
        ELSIF NOT __ISVALIDREF(inoConfig) THEN
            _varInfo := __VARINFO(inoConfig);
            Messenger.Programming(_sb.Clear().Append('<#Invalid reference: #>').Append(_varInfo.Symbol).ToString()).Pin();
        ELSIF NOT __ISVALIDREF(inoStatus) THEN
            _varInfo := __VARINFO(inoStatus);
            Messenger.Programming(_sb.Clear().Append('<#Invalid reference: #>').Append(_varInfo.Symbol).ToString()).Pin();
        ELSE
            _progress := _progress + 1;
        END_IF
    END_IF

    IF _progress = 1 THEN
        CallTimers(FALSE);

        IF _jobName = '' THEN
            Messenger.Programming('<#Empty job name inserted!#>').Pin();
            THIS^.ThrowWhen(TRUE);
        ELSE
            _progress := _progress + 1;
        END_IF
    END_IF

    IF _progress = 2 THEN
        THIS^.inoStatus.ActionDescription :=
            _sb.Clear().Append('<#Change job by name (').Append(THIS^._jobName).Append(') is running.#>').ToString();

        THIS^.Messenger.OnCondition(_infoTimer.Q).Warning('<#Waiting for the signal CommandExecuting to be reseted!#>').Pin();
        THIS^.inoIoData.InspectionControl.ExecuteCommand := FALSE;
        THIS^.inoIoData.InspectionControl.ClearError := FALSE;
        THIS^.inoIoData.AcquisitionControl.SetOffline := FALSE;

        IF NOT THIS^.inoIoData.InspectionStatus.CommandExecuting THEN
            CallTimers(FALSE);
            _progress := _progress + 1;
        END_IF
    END_IF

    IF _progress = 3 THEN
        THIS^.Messenger.OnCondition(_infoTimer.Q).Warning('<#Waiting for the signal Online to be reseted!#>').Pin();
        THIS^.inoIoData.AcquisitionControl.SetOffline := TRUE;

        IF (NOT THIS^.inoIoData.AcquisitionStatus.Online) THEN
            CallTimers(FALSE);
            _progress := _progress + 1;
        END_IF
    END_IF

    IF _progress = 4 THEN
        THIS^.Messenger.OnCondition(_infoTimer.Q).Warning('<#Waiting for the signal Error to be reseted!#>').Pin();
        THIS^.inoIoData.AcquisitionControl.SetOffline := TRUE;
        THIS^.inoIoData.InspectionControl.ExecuteCommand := FALSE;
        THIS^.inoIoData.InspectionControl.ClearError := THIS^.inoIoData.InspectionStatus.Error;

        IF NOT THIS^.inoIoData.InspectionStatus.Error THEN
            CallTimers(FALSE);
            _progress := _progress + 1;
        END_IF
    END_IF

    IF _progress = 5 THEN
        THIS^.Messenger.OnCondition(_infoTimer.Q).Warning('<#Waiting for the Job name to be written to the User data!#>').Pin();
        THIS^.inoIoData.AcquisitionControl.SetOffline := TRUE;

        IF SetUserDataAsString(_jobName, 0) THEN
            CallTimers(FALSE);
            _progress := _progress + 1;
        END_IF
    END_IF

    IF _progress = 6 THEN
        THIS^.Messenger.OnCondition(_infoTimer.Q).Warning('<#Waiting for the signal ExtendedUserDataSetAcknowledge to be set!#>').Pin();
        THIS^.inoIoData.AcquisitionControl.SetOffline := TRUE;
        THIS^.inoIoData.InspectionControl.ExtendedUserDataSet := TRUE;

        IF (THIS^.inoIoData.InspectionStatus.ExtendedUserDataSetAcknowledge) THEN
            CallTimers(FALSE);
            _progress := _progress + 1;
        END_IF
    END_IF

    IF _progress = 7 THEN
        THIS^.Messenger.OnCondition(_infoTimer.Q).Warning('<#Waiting for the signal ExtendedUserDataSetAcknowledge to be reseted!#>').Pin();
        THIS^.inoIoData.AcquisitionControl.SetOffline := TRUE;
        THIS^.inoIoData.InspectionControl.ExtendedUserDataSet := FALSE;

        IF (NOT THIS^.inoIoData.InspectionStatus.ExtendedUserDataSetAcknowledge) THEN
            CallTimers(FALSE);
            _progress := _progress + 1;
        END_IF
    END_IF

    IF _progress = 8 THEN
        THIS^.Messenger.OnCondition(_infoTimer.Q).Warning('<#Waiting for the signal CommandComplete to be set!#>').Pin();
        THIS^.inoIoData.AcquisitionControl.SetOffline := TRUE;
        THIS^.inoIoData.CommandControl.Command := 16#4000;
        THIS^.inoIoData.InspectionControl.ExecuteCommand := TRUE;

        IF (THIS^.inoIoData.InspectionStatus.CommandComplete AND NOT THIS^.inoIoData.InspectionStatus.CommandFailed) THEN
            CallTimers(FALSE);
            _progress := _progress + 1;
        ELSIF (THIS^.inoIoData.InspectionStatus.CommandComplete AND
            THIS^.inoIoData.InspectionStatus.CommandFailed AND
            NOT THIS^.inoIoData.InspectionStatus.CommandExecuting) THEN
            _progress := 20;
        END_IF;
    END_IF

    IF _progress = 9 THEN
        THIS^.Messenger.OnCondition(_infoTimer.Q).Warning('<#Waiting for the signal CommandComplete to be reseted!#>').Pin();
        THIS^.inoIoData.AcquisitionControl.SetOffline := TRUE;
        THIS^.inoIoData.CommandControl.Command := 0;
        THIS^.inoIoData.InspectionControl.ExecuteCommand := FALSE;

        IF (NOT THIS^.inoIoData.InspectionStatus.CommandComplete) THEN
            CallTimers(FALSE);
            _progress := _progress + 1;
        END_IF;
    END_IF

    IF _progress = 10 THEN
        THIS^.Messenger.OnCondition(_infoTimer.Q).Warning('<#Waiting for the signal Online to be set!#>').Pin();
        THIS^.inoIoData.AcquisitionControl.SetOffline := FALSE;

        IF (THIS^.inoIoData.AcquisitionStatus.Online) THEN
            CallTimers(FALSE);
            _progress := _progress + 1;
        END_IF
    END_IF

    IF _progress = 11 THEN
        THIS^.inoStatus.CurrentJobName := _jobName;
        THIS^.inoIoData.InspectionControl.ExecuteCommand := FALSE;
        THIS^.inoIoData.AcquisitionControl.SetOffline := FALSE;
        THIS^.inoIoData.InspectionControl.ClearError := FALSE;
        THIS^.inoIoData.CommandControl.Command := 0;
        THIS^.ThrowWhen(FALSE);
        THIS^.DoneWhen(TRUE);
        _progress := 0;
    END_IF

    IF _progress = 20 THEN
        Messenger.Error(CONCAT('<#Change job by name failed. Error code:#>', UINT_TO_STRING(inoIoData.InspectionStatus.ErrorCode))).Pin();
        THIS^.inoIoData.InspectionControl.ExecuteCommand := FALSE;
        THIS^.inoIoData.AcquisitionControl.SetOffline := FALSE;
        THIS^.inoIoData.CommandControl.Command := 0;
        THIS^.ThrowWhen(TRUE);
        THIS^.DoneWhen(FALSE);
    END_IF

    CallTimers(TRUE);
    THIS^.ThrowWhen(_errorTimer.Q);
END_IF

METHOD CallTimers
VAR_INPUT
    inValue : BOOL;
END_VAR
_infoTimer(IN := inValue, PT := THIS^.inoConfig.InfoTime);
_errorTimer(IN := inValue, PT := THIS^.inoConfig.ErrorTime);
END_METHOD

{attribute 'hide'}
METHOD PUBLIC FB_init : BOOL
VAR_INPUT
    bInitRetains : BOOL; // if TRUE, the retain variables are initialized (warm start / cold start)
    bInCopyCode : BOOL; // if TRUE, the instance afterwards gets moved into the copy code (online change)
    ParentObject : ITcoObject;
END_VAR
END_METHOD

METHOD INTERNAL InvokeWithParameters : ITcoTaskStatus
VAR_INPUT
    inJobName : STRING;
END_VAR
_jobName := inJobName;
InvokeWithParameters := THIS^.Invoke();
END_METHOD

(*~
    <docu>
        <summary>
            Executes when task is aborted.
        </summary>
    </docu>
~*)
METHOD PROTECTED OnAbort
THIS^.inoStatus.ActionDescription :=
    _sb.Clear().Append('<#Change job by name (').Append(THIS^._jobName).Append(') aborted, while not yet finished.#>').ToString();
END_METHOD

(*~
    <docu>
        <summary>
            Executes when task reaches the ```Done``` state .
        </summary>
    </docu>
~*)
METHOD PROTECTED OnDone
THIS^.inoStatus.ActionDescription :=
    _sb.Clear().Append('<#Change job by name (').Append(THIS^._jobName).Append(') was completed succesfully.#>').ToString();
END_METHOD

(*~
    <docu>
        <summary>
            Executes when task reaches the ```Error``` state.
            <para>
                Do not confuse with <see cref="PlcDocu.TcoCore.TcoTask.WhileError()"/>, that is called cyclically until '''Error''' state is left.
            </para>
        </summary>
    </docu>
~*)
METHOD PROTECTED OnError
THIS^.inoStatus.ActionDescription :=
    _sb.Clear().Append('<#Change job by name (').Append(THIS^._jobName).Append(') finished with error.#>').ToString();
END_METHOD

METHOD PROTECTED OnStart
THIS^.inoStatus.ActionDescription := _sb.Clear().Append('<#Change job by name (').Append(THIS^._jobName).Append(') started.#>').ToString();
END_METHOD

(*~
    <docu>
        <summary>
            Restores this instance to the Ready state. Can be called explicitly or from within one of the restore mechanisms.
            <para>
                See also <see cref="PlcDocu.TcoCore.TcoTask.AutoRestorable()"/>
            </para>
        </summary>
    </docu>
~*)
METHOD Restore : ITcoRestorable
SUPER^.Restore();
_progress := 0;
CallTimers(FALSE);
Messenger.UnPin();
END_METHOD

METHOD INTERNAL SetUserDataAsString : BOOL
VAR_INPUT
    inValue : STRING;
    inPosition : UINT;
END_VAR
VAR
    _index : UINT;
    _size : UINT;
    _bufferSize : UINT;
END_VAR
SetUserDataAsString := FALSE;
_size := LEN(inValue);
//_bufferSize := SIZEOF(inoUserData.UserData)/SIZEOF(inoUserData.UserData[0]);
_bufferSize := SIZEOF(THIS^.inoIoData.UserData.UserData) / SIZEOF(THIS^.inoIoData.UserData.UserData[0]);

IF (inPosition + _size) > THIS^.inoConfig.UserDataSize THEN
    Messenger.Programming('<#Index of UserData in method SetUserDataAsString exceeds the size hardware structure mapped!#>');
    RETURN;
END_IF

IF (inPosition + _size) > _bufferSize THEN
    Messenger.Programming('<#Index of UserData in method SetUserDataAsString exceeds the defined size!#>');
    RETURN;
END_IF

FOR _index := 1 TO _size BY 1 DO
    THIS^.inoIoData.UserData.UserData[inPosition + _index - 1] := F_ToASC(MID(inValue, 1, _index));
END_FOR;

FOR _index := inPosition + _size TO _bufferSize BY 1 DO
    THIS^.inoIoData.UserData.UserData[_index] := 0;
END_FOR;

SetUserDataAsString := TRUE;
END_METHOD

END_FUNCTION_BLOCK

// ---- POUs/TcoInsight/v_5_x_x/Tasks/TcoInsightChangeJobByNumber_v_5_x_x.TcPOU
FUNCTION_BLOCK TcoInsightChangeJobByNumber_v_5_x_x EXTENDS TcoCore.TcoTask
VAR_IN_OUT
    inoIoData : TcoInsightIO_v_5_x_x;
    inoConfig : TcoInsightConfig_v_5_x_x;
    inoStatus : TcoInsightStatus_v_5_x_x;
END_VAR
VAR
    {attribute addProperty Name "<#Job number#>"}
    _jobNumber : UINT;
END_VAR
VAR
    {attribute 'hide'}
    _progress : INT := 0;
    {attribute 'hide'}
    _infoTimer : TON;
    {attribute 'hide'}
    _errorTimer : TON;
    {attribute 'hide'}
    _varInfo : __SYSTEM.VAR_INFO;
    {attribute 'hide'}
    _sb : TcoCore.StringBuilder;
END_VAR

IF Execute() THEN
    IF _progress = 0 THEN
        IF NOT __ISVALIDREF(inoIoData) THEN
            _varInfo := __VARINFO(inoIoData);
            Messenger.Programming(_sb.Clear().Append('<#Invalid reference: #>').Append(_varInfo.Symbol).ToString()).Pin();
        ELSIF NOT __ISVALIDREF(inoConfig) THEN
            _varInfo := __VARINFO(inoConfig);
            Messenger.Programming(_sb.Clear().Append('<#Invalid reference: #>').Append(_varInfo.Symbol).ToString()).Pin();
        ELSIF NOT __ISVALIDREF(inoStatus) THEN
            _varInfo := __VARINFO(inoStatus);
            Messenger.Programming(_sb.Clear().Append('<#Invalid reference: #>').Append(_varInfo.Symbol).ToString()).Pin();
        ELSE
            _progress := _progress + 1;
        END_IF
    END_IF

    IF _progress = 1 THEN
        CallTimers(FALSE);

